C05482=1223.178,35.785,-43.751,-179.162,5.442,148.698
C05483=1223.173,36.035,-43.767,-179.159,5.442,148.697
C05484=1223.168,36.285,-43.783,-179.156,5.443,148.696
C05485=1223.163,36.534,-43.798,-179.154,5.443,148.696
C05486=1223.158,36.784,-43.815,-179.151,5.444,148.695
C05487=1223.154,37.033,-43.830,-179.148,5.444,148.694
C05488=1223.148,37.282,-43.846,-179.146,5.445,148.694
C05489=1223.144,37.532,-43.862,-179.144,5.445,148.693
C05490=1223.138,37.781,-43.878,-179.142,5.446,148.692
C05491=1223.134,38.031,-43.894,-179.139,5.446,148.692
C05492=1223.128,38.280,-43.910,-179.136,5.447,148.691
C05493=1223.123,38.529,-43.926,-179.134,5.447,148.690
C05494=1223.119,38.779,-43.942,-179.131,5.448,148.690
C05495=1223.113,39.028,-43.958,-179.128,5.448,148.689
C05496=1223.108,39.278,-43.974,-179.126,5.449,148.688
C05497=1223.103,39.527,-43.990,-179.124,5.450,148.688
C05498=1223.099,39.777,-44.006,-179.121,5.450,148.687
C05499=1223.093,40.026,-44.022,-179.118,5.451,148.687
C05500=1223.089,40.275,-44.037,-179.116,5.451,148.686
C05501=1223.084,40.525,-44.053,-179.114,5.451,148.685
C05502=1223.079,40.774,-44.070,-179.111,5.452,148.685
C05503=1223.074,41.024,-44.086,-179.108,5.452,148.684
C05504=1223.069,41.273,-44.102,-179.106,5.453,148.683
C05505=1223.064,41.523,-44.118,-179.104,5.454,148.683
C05506=1223.059,41.772,-44.134,-179.101,5.454,148.682
C05507=1223.054,42.022,-44.150,-179.098,5.455,148.681
C05508=1223.049,42.271,-44.166,-179.096,5.455,148.681
C05509=1223.045,42.521,-44.182,-179.093,5.456,148.680
C05510=1223.039,42.770,-44.199,-179.090,5.457,148.679
C05511=1223.035,43.020,-44.215,-179.088,5.457,148.679
C05512=1223.030,43.268,-44.231,-179.085,5.458,148.678
C05513=1223.025,43.519,-44.247,-179.083,5.459,148.678
C05514=1223.019,43.768,-44.264,-179.081,5.458,148.677
C05515=1223.014,44.018,-44.280,-179.078,5.459,148.676
C05516=1223.009,44.267,-44.296,-179.076,5.459,148.676
C05517=1223.005,44.516,-44.313,-179.073,5.460,148.675
C05518=1222.999,44.765,-44.328,-179.070,5.461,148.674
C05519=1222.995,45.015,-44.345,-179.068,5.461,148.674
C05520=1222.989,45.264,-44.361,-179.065,5.462,148.673
C05521=1222.985,45.514,-44.377,-179.063,5.463,148.672
C05522=1222.980,45.763,-44.394,-179.060,5.463,148.672
C05523=1222.975,46.013,-44.410,-179.058,5.464,148.671
C05524=1222.970,46.261,-44.426,-179.055,5.464,148.670
C05525=1222.965,46.512,-44.442,-179.052,5.465,148.670
C05526=1222.960,46.760,-44.458,-179.050,5.465,148.669
C05527=1222.955,47.010,-44.475,-179.047,5.466,148.668
C05528=1222.949,47.260,-44.491,-179.045,5.467,148.668
C05529=1222.945,47.509,-44.508,-179.042,5.467,148.667
C05530=1222.941,47.758,-44.524,-179.040,5.468,148.667
C05531=1222.935,48.008,-44.540,-179.038,5.468,148.666
C05532=1222.931,48.257,-44.557,-179.035,5.468,148.665
C05533=1222.926,48.506,-44.573,-179.032,5.469,148.665
C05534=1222.920,48.756,-44.590,-179.030,5.469,148.664
C05535=1222.915,49.005,-44.606,-179.027,5.470,148.663
C05536=1222.911,49.255,-44.622,-179.025,5.471,148.663
C05537=1222.906,49.504,-44.639,-179.022,5.471,148.662
C05538=1222.901,49.753,-44.655,-179.020,5.472,148.661
C05539=1222.896,50.003,-44.671,-179.017,5.473,148.661
C05540=1222.890,50.252,-44.688,-179.014,5.473,148.660
C05541=1222.886,50.502,-44.705,-179.012,5.474,148.659
C05542=1222.881,50.751,-44.722,-179.010,5.475,148.659
C05543=1222.876,51.001,-44.737,-179.007,5.475,148.658
C05544=1222.872,51.250,-44.754,-179.004,5.476,148.658
C05545=1222.866,51.499,-44.771,-179.002,5.476,148.657
C05546=1222.861,51.749,-44.787,-178.999,5.477,148.656
C05547=1222.857,51.998,-44.804,-178.996,5.477,148.656
C05548=1222.851,52.248,-44.820,-178.994,5.478,148.655
C05549=1222.847,52.497,-44.836,-178.992,5.479,148.655
C05550=1222.842,52.747,-44.854,-178.989,5.479,148.654
C05551=1222.837,52.996,-44.870,-178.986,5.480,148.653
C05552=1222.832,53.245,-44.887,-178.984,5.481,148.653
C05553=1222.828,53.495,-44.903,-178.981,5.481,148.652
C05554=1222.822,53.744,-44.920,-178.978,5.482,148.651
C05555=1222.817,53.994,-44.936,-178.976,5.483,148.651
C05556=1222.812,54.243,-44.952,-178.974,5.483,148.650
C05557=1222.807,54.492,-44.970,-178.971,5.484,148.649
C05558=1222.802,54.742,-44.986,-178.968,5.484,148.649
C05559=1222.797,54.991,-45.003,-178.966,5.485,148.648
C05560=1222.792,55.260,-45.021,-178.963,5.485,148.647
C05561=1222.787,55.527,-45.039,-178.960,5.486,148.647
C05562=1222.782,55.797,-45.056,-178.958,5.487,148.646
C05563=1222.776,56.065,-45.075,-178.955,5.487,148.645
C05564=1222.771,56.314,-45.091,-178.953,5.488,148.645
C05565=1222.767,56.564,-45.108,-178.950,5.488,148.644
C05566=1222.761,56.813,-45.125,-178.948,5.489,148.644
C05567=1222.756,57.062,-45.142,-178.945,5.490,148.643
C05568=1222.752,57.312,-45.158,-178.942,5.490,148.642
C05569=1222.747,57.562,-45.176,-178.940,5.491,148.642
C05570=1222.742,57.810,-45.192,-178.937,5.491,148.641
C05571=1222.736,58.060,-45.209,-178.935,5.492,148.640
C05572=1222.732,58.310,-45.226,-178.932,5.493,148.640
C05573=1222.727,58.558,-45.242,-178.930,5.494,148.639
C05574=1222.722,58.808,-45.259,-178.927,5.494,148.639
C05575=1222.717,59.058,-45.276,-178.925,5.495,148.638
C05576=1222.712,59.308,-45.293,-178.922,5.495,148.637
C05577=1222.707,59.556,-45.310,-178.920,5.496,148.637
C05578=1222.703,59.805,-45.327,-178.917,5.497,148.636
C05579=1222.697,60.055,-45.344,-178.914,5.497,148.635
C05580=1222.693,60.304,-45.361,-178.912,5.498,148.635
C05581=1222.687,60.554,-45.378,-178.909,5.498,148.634
C05582=1222.683,60.803,-45.394,-178.907,5.499,148.633
C05583=1222.677,61.053,-45.412,-178.904,5.500,148.633
C05584=1222.673,61.302,-45.428,-178.902,5.501,148.632
C05585=1222.668,61.551,-45.445,-178.899,5.501,148.632
C05586=1222.663,61.800,-45.463,-178.897,5.502,148.631
C05587=1222.658,62.050,-45.479,-178.894,5.502,148.630
C05588=1222.653,62.300,-45.497,-178.892,5.503,148.630
C05589=1222.649,62.549,-45.513,-178.889,5.504,148.629
C05590=1222.643,62.798,-45.530,-178.886,5.504,148.629
C05591=1222.639,63.047,-45.548,-178.884,5.505,148.628
C05592=1222.633,63.297,-45.565,-178.881,5.505,148.627
C05593=1222.629,63.546,-45.582,-178.879,5.506,148.627
C05594=1222.624,63.796,-45.599,-178.876,5.507,148.626
C05595=1222.619,64.045,-45.615,-178.874,5.508,148.626
C05596=1222.614,64.294,-45.633,-178.871,5.508,148.625
C05597=1222.609,64.544,-45.650,-178.869,5.509,148.624
C05598=1222.604,64.793,-45.667,-178.866,5.510,148.624
C05599=1222.599,65.043,-45.684,-178.863,5.511,148.623
C05600=1222.594,65.291,-45.701,-178.861,5.512,148.622
C05601=1222.589,65.541,-45.719,-178.858,5.512,148.622
C05602=1222.584,65.791,-45.735,-178.855,5.513,148.621
C05603=1222.580,66.040,-45.753,-178.853,5.514,148.621
C05604=1222.575,66.289,-45.770,-178.851,5.514,148.620
C05605=1222.570,66.539,-45.787,-178.848,5.515,148.619
C05606=1222.566,66.788,-45.805,-178.845,5.515,148.619
C05607=1222.560,67.037,-45.821,-178.843,5.516,148.618
C05608=1222.555,67.287,-45.839,-178.841,5.517,148.618
C05609=1222.550,67.536,-45.856,-178.838,5.517,148.617
C05610=1222.545,67.785,-45.873,-178.835,5.518,148.616
C05611=1222.541,68.035,-45.890,-178.833,5.519,148.616
C05612=1222.536,68.284,-45.908,-178.830,5.519,148.615
C05613=1222.531,68.534,-45.925,-178.828,5.520,148.615
C05614=1222.526,68.783,-45.942,-178.825,5.521,148.614
C05615=1222.521,69.032,-45.960,-178.823,5.521,148.613
C05616=1222.515,69.282,-45.977,-178.820,5.522,148.613
C05617=1222.511,69.530,-45.994,-178.818,5.523,148.612
C05618=1222.506,69.780,-46.011,-178.815,5.523,148.611
C05619=1222.501,70.029,-46.029,-178.813,5.524,148.611
C05620=1222.497,70.279,-46.046,-178.809,5.525,148.610
C05621=1222.491,70.529,-46.063,-178.807,5.526,148.609
C05622=1222.486,70.778,-46.081,-178.805,5.527,148.609
C05623=1222.482,71.027,-46.098,-178.802,5.527,148.608
C05624=1222.477,71.277,-46.116,-178.799,5.528,148.608
C05625=1222.471,71.526,-46.133,-178.797,5.529,148.607
C05626=1222.467,71.775,-46.150,-178.795,5.530,148.607
C05627=1222.462,72.024,-46.168,-178.792,5.530,148.606
C05628=1222.457,72.273,-46.186,-178.789,5.531,148.605
C05629=1222.452,72.523,-46.202,-178.787,5.531,148.605
C05630=1222.448,72.772,-46.220,-178.785,5.532,148.604
C05631=1222.442,73.022,-46.237,-178.782,5.533,148.604
C05632=1222.437,73.271,-46.255,-178.779,5.533,148.603
C05633=1222.433,73.520,-46.273,-178.777,5.534,148.602
C05634=1222.428,73.770,-46.290,-178.774,5.535,148.602
C05635=1222.423,74.019,-46.308,-178.771,5.536,148.601
C05636=1222.418,74.269,-46.325,-178.769,5.537,148.601
C05637=1222.414,74.518,-46.343,-178.766,5.537,148.600
C05638=1222.409,74.767,-46.361,-178.763,5.538,148.599
C05639=1222.404,75.017,-46.378,-178.761,5.539,148.599
C05640=1222.399,75.266,-46.396,-178.759,5.540,148.598
C05641=1222.393,75.516,-46.413,-178.756,5.540,148.597
C05642=1222.389,75.764,-46.431,-178.753,5.541,148.597
C05643=1222.384,76.014,-46.449,-178.751,5.542,148.596
C05644=1222.379,76.263,-46.466,-178.749,5.542,148.596
C05645=1222.374,76.513,-46.484,-178.746,5.543,148.595
C05646=1222.369,76.762,-46.502,-178.743,5.543,148.594
C05647=1222.365,77.011,-46.518,-178.741,5.545,148.594
C05648=1222.360,77.260,-46.536,-178.738,5.546,148.593
C05649=1222.355,77.510,-46.554,-178.735,5.546,148.593
C05650=1222.350,77.759,-46.572,-178.733,5.547,148.592
C05651=1222.345,78.009,-46.590,-178.731,5.548,148.592
C05652=1222.340,78.258,-46.608,-178.728,5.548,148.591
C05653=1222.335,78.507,-46.626,-178.725,5.549,148.590
C05654=1222.331,78.756,-46.642,-178.723,5.550,148.590
C05655=1222.326,79.006,-46.660,-178.721,5.551,148.589
C05656=1222.321,79.255,-46.678,-178.718,5.551,148.589
C05657=1222.316,79.504,-46.696,-178.715,5.553,148.588
C05658=1222.311,79.754,-46.713,-178.712,5.553,148.587
C05659=1222.306,80.003,-46.731,-178.710,5.554,148.587
C05660=1222.301,80.252,-46.749,-178.708,5.555,148.586
C05661=1222.296,80.501,-46.767,-178.705,5.555,148.585
C05662=1222.291,80.750,-46.785,-178.703,5.556,148.585
C05663=1222.286,81.001,-46.803,-178.700,5.557,148.584
C05664=1222.281,81.268,-46.822,-178.697,5.558,148.584
C05665=1222.276,81.537,-46.841,-178.694,5.559,148.583
C05666=1222.271,81.805,-46.861,-178.692,5.559,148.582
C05667=1222.265,82.074,-46.880,-178.689,5.560,148.582
C05668=1222.260,82.323,-46.898,-178.686,5.561,148.581
C05669=1222.255,82.572,-46.916,-178.684,5.562,148.581
C05670=1222.251,82.822,-46.934,-178.681,5.563,148.580
C05671=1222.246,83.071,-46.952,-178.678,5.564,148.579
C05672=1222.241,83.320,-46.970,-178.676,5.564,148.579
C05673=1222.236,83.570,-46.988,-178.674,5.565,148.578
C05674=1222.231,83.819,-47.006,-178.671,5.566,148.578
C05675=1222.226,84.068,-47.024,-178.668,5.566,148.577
C05676=1222.222,84.317,-47.042,-178.666,5.567,148.577
C05677=1222.216,84.567,-47.059,-178.663,5.569,148.576
C05678=1222.212,84.817,-47.077,-178.661,5.569,148.575
C05679=1222.207,85.066,-47.095,-178.658,5.570,148.575
C05680=1222.202,85.315,-47.113,-178.656,5.571,148.574
C05681=1222.197,85.564,-47.131,-178.653,5.571,148.574
C05682=1222.192,85.814,-47.149,-178.651,5.572,148.573
C05683=1222.187,86.063,-47.167,-178.648,5.573,148.572
C05684=1222.183,86.312,-47.185,-178.645,5.574,148.572
C05685=1222.178,86.562,-47.204,-178.643,5.575,148.571
C05686=1222.173,86.811,-47.222,-178.640,5.575,148.571
C05687=1222.168,87.060,-47.240,-178.638,5.576,148.570
C05688=1222.163,87.309,-47.258,-178.635,5.577,148.569
C05689=1222.159,87.558,-47.276,-178.633,5.578,148.569
C05690=1222.154,87.807,-47.294,-178.630,5.579,148.568
C05691=1222.150,88.057,-47.313,-178.627,5.580,148.568
C05692=1222.144,88.306,-47.331,-178.625,5.581,148.567
C05693=1222.139,88.556,-47.349,-178.623,5.581,148.567
C05694=1222.134,88.805,-47.367,-178.620,5.582,148.566
C05695=1222.129,89.054,-47.385,-178.617,5.583,148.565
C05696=1222.125,89.304,-47.403,-178.615,5.583,148.565
C05697=1222.120,89.553,-47.421,-178.612,5.585,148.564
C05698=1222.115,89.802,-47.439,-178.609,5.586,148.564
C05699=1222.110,90.051,-47.459,-178.607,5.586,148.563
C05700=1222.105,90.300,-47.477,-178.605,5.587,148.563
C05701=1222.101,90.550,-47.495,-178.602,5.588,148.562
C05702=1222.096,90.799,-47.513,-178.599,5.588,148.561
C05703=1222.091,91.048,-47.531,-178.597,5.590,148.561
C05704=1222.086,91.298,-47.549,-178.594,5.591,148.560
C05705=1222.081,91.547,-47.569,-178.591,5.591,148.560
C05706=1222.076,91.796,-47.587,-178.589,5.592,148.559
C05707=1222.071,92.045,-47.605,-178.587,5.593,148.558
C05708=1222.066,92.295,-47.623,-178.584,5.593,148.558
C05709=1222.062,92.545,-47.641,-178.581,5.595,148.557
C05710=1222.057,92.793,-47.660,-178.579,5.596,148.557
C05711=1222.052,93.043,-47.678,-178.576,5.596,148.556
C05712=1222.047,93.292,-47.696,-178.574,5.597,148.556
C05713=1222.043,93.542,-47.714,-178.571,5.598,148.555
C05714=1222.037,93.790,-47.734,-178.569,5.599,148.554
C05715=1222.032,94.040,-47.752,-178.566,5.600,148.554
C05716=1222.028,94.290,-47.770,-178.563,5.601,148.553
C05717=1222.023,94.538,-47.789,-178.561,5.602,148.553
C05718=1222.018,94.788,-47.807,-178.558,5.602,148.552
C05719=1222.013,95.037,-47.825,-178.556,5.603,148.552
C05720=1222.009,95.286,-47.844,-178.553,5.604,148.551
C05721=1222.004,95.535,-47.862,-178.550,5.605,148.550
C05722=1221.998,95.785,-47.881,-178.548,5.606,148.550
C05723=1221.994,96.034,-47.900,-178.545,5.607,148.549
C05724=1221.989,96.283,-47.918,-178.543,5.607,148.549
C05725=1221.984,96.533,-47.937,-178.540,5.609,148.548
C05726=1221.980,96.782,-47.956,-178.538,5.610,148.548
C05727=1221.975,97.031,-47.974,-178.535,5.611,148.547
C05728=1221.969,97.280,-47.993,-178.533,5.611,148.546
C05729=1221.965,97.530,-48.011,-178.530,5.612,148.546
C05730=1221.960,97.779,-48.029,-178.527,5.614,148.545
C05731=1221.955,98.028,-48.049,-178.525,5.614,148.545
C05732=1221.951,98.278,-48.067,-178.522,5.615,148.544
C05733=1221.946,98.526,-48.086,-178.520,5.616,148.544
C05734=1221.940,98.776,-48.104,-178.517,5.616,148.543
C05735=1221.936,99.025,-48.123,-178.514,5.618,148.542
C05736=1221.931,99.274,-48.141,-178.512,5.619,148.542
C05737=1221.926,99.523,-48.160,-178.510,5.619,148.541
C05738=1221.922,99.773,-48.179,-178.507,5.620,148.541
C05739=1221.916,100.022,-48.198,-178.505,5.621,148.540
C05740=1221.912,100.272,-48.216,-178.502,5.622,148.540
C05741=1221.907,100.520,-48.235,-178.499,5.623,148.539
C05742=1221.902,100.770,-48.254,-178.497,5.624,148.539
C05743=1221.898,101.019,-48.273,-178.494,5.624,148.538
C05744=1221.892,101.268,-48.291,-178.492,5.626,148.538
C05745=1221.888,101.518,-48.310,-178.489,5.627,148.537
C05746=1221.883,101.767,-48.329,-178.486,5.627,148.536
C05747=1221.878,102.016,-48.348,-178.484,5.628,148.536
C05748=1221.874,102.265,-48.367,-178.482,5.629,148.535
C05749=1221.868,102.514,-48.385,-178.478,5.630,148.535
C05750=1221.864,102.764,-48.404,-178.476,5.631,148.534
C05751=1221.859,103.013,-48.423,-178.474,5.632,148.533
C05752=1221.854,103.262,-48.442,-178.471,5.633,148.533
C05753=1221.849,103.511,-48.461,-178.468,5.634,148.532
C05754=1221.844,103.761,-48.479,-178.466,5.635,148.532
C05755=1221.840,104.010,-48.499,-178.464,5.636,148.531
C05756=1221.835,104.259,-48.518,-178.461,5.637,148.531
C05757=1221.830,104.509,-48.537,-178.458,5.638,148.530
C05758=1221.825,104.757,-48.555,-178.456,5.639,148.530
C05759=1221.821,105.007,-48.575,-178.453,5.639,148.529
C05760=1221.816,105.256,-48.593,-178.450,5.640,148.528
C05761=1221.810,105.505,-48.612,-178.448,5.642,148.528
C05762=1221.806,105.755,-48.632,-178.445,5.642,148.527
C05763=1221.801,106.004,-48.650,-178.443,5.643,148.527
C05764=1221.796,106.253,-48.669,-178.440,5.644,148.526
C05765=1221.791,106.502,-48.688,-178.437,5.645,148.526
C05766=1221.787,106.751,-48.708,-178.435,5.646,148.525
C05767=1221.782,107.001,-48.726,-178.433,5.647,148.525
C05768=1221.777,107.269,-48.747,-178.430,5.648,148.524
C05769=1221.771,107.537,-48.768,-178.427,5.649,148.524
C05770=1221.766,107.806,-48.788,-178.425,5.650,148.523
C05771=1221.761,108.074,-48.809,-178.421,5.651,148.522
C05772=1221.757,108.324,-48.828,-178.419,5.652,148.522
C05773=1221.751,108.573,-48.847,-178.417,5.653,148.521
C05774=1221.747,108.822,-48.865,-178.414,5.654,148.521
C05775=1221.742,109.071,-48.885,-178.411,5.655,148.520
C05776=1221.737,109.321,-48.904,-178.409,5.656,148.520
C05777=1221.732,109.569,-48.923,-178.406,5.657,148.519
C05778=1221.727,109.819,-48.943,-178.403,5.658,148.518
C05779=1221.723,110.069,-48.962,-178.401,5.659,148.518
C05780=1221.718,110.317,-48.981,-178.399,5.660,148.517
C05781=1221.713,110.567,-49.001,-178.396,5.661,148.517
C05782=1221.708,110.816,-49.019,-178.393,5.662,148.516
C05783=1221.704,111.065,-49.038,-178.391,5.663,148.516
C05784=1221.698,111.314,-49.058,-178.388,5.664,148.515
C05785=1221.694,111.564,-49.077,-178.386,5.665,148.515
C05786=1221.689,111.812,-49.096,-178.383,5.666,148.514
C05787=1221.684,112.062,-49.116,-178.380,5.667,148.513
C05788=1221.679,112.312,-49.135,-178.378,5.668,148.513
C05789=1221.675,112.560,-49.154,-178.375,5.669,148.512
C05790=1221.670,112.810,-49.174,-178.373,5.670,148.512
C05791=1221.665,113.059,-49.193,-178.370,5.671,148.511
C05792=1221.660,113.308,-49.213,-178.368,5.672,148.511
C05793=1221.655,113.557,-49.231,-178.365,5.673,148.510
C05794=1221.651,113.806,-49.251,-178.362,5.674,148.510
C05795=1221.646,114.056,-49.271,-178.360,5.675,148.509
C05796=1221.641,114.305,-49.290,-178.357,5.676,148.509
C05797=1221.637,114.554,-49.309,-178.355,5.677,148.508
C05798=1221.632,114.804,-49.329,-178.352,5.678,148.508
C05799=1221.627,115.052,-49.348,-178.350,5.679,148.507
C05800=1221.622,115.302,-49.368,-178.347,5.680,148.506
C05801=1221.616,115.551,-49.387,-178.344,5.681,148.506
C05802=1221.612,115.800,-49.406,-178.342,5.682,148.505
C05803=1221.608,116.050,-49.426,-178.339,5.683,148.505
C05804=1221.602,116.299,-49.445,-178.337,5.684,148.504
C05805=1221.598,116.547,-49.465,-178.334,5.685,148.504
C05806=1221.593,116.797,-49.485,-178.332,5.686,148.503
C05807=1221.588,117.046,-49.504,-178.329,5.687,148.503
C05808=1221.584,117.295,-49.523,-178.326,5.688,148.502
C05809=1221.579,117.545,-49.543,-178.324,5.689,148.502
C05810=1221.574,117.794,-49.562,-178.321,5.690,148.501
C05811=1221.569,118.043,-49.582,-178.319,5.691,148.501
C05812=1221.565,118.292,-49.602,-178.316,5.692,148.500
C05813=1221.559,118.541,-49.622,-178.314,5.693,148.500
C05814=1221.554,118.791,-49.641,-178.311,5.694,148.499
C05815=1221.550,119.040,-49.660,-178.308,5.696,148.499
C05816=1221.545,119.289,-49.680,-178.306,5.696,148.498
C05817=1221.541,119.538,-49.700,-178.304,5.697,148.498
C05818=1221.536,119.787,-49.720,-178.301,5.699,148.497
C05819=1221.531,120.036,-49.739,-178.298,5.699,148.496
C05820=1221.526,120.286,-49.758,-178.296,5.700,148.496
C05821=1221.521,120.535,-49.779,-178.293,5.702,148.495
C05822=1221.516,120.783,-49.798,-178.291,5.703,148.495
C05823=1221.511,121.033,-49.818,-178.288,5.703,148.494
C05824=1221.507,121.283,-49.837,-178.285,5.705,148.494
C05825=1221.502,121.532,-49.858,-178.283,5.706,148.493
C05826=1221.497,121.780,-49.877,-178.281,5.707,148.493
C05827=1221.492,122.030,-49.897,-178.277,5.708,148.492
C05828=1221.488,122.279,-49.917,-178.275,5.709,148.492
C05829=1221.484,122.528,-49.936,-178.273,5.710,148.491
C05830=1221.478,122.777,-49.956,-178.270,5.712,148.491
C05831=1221.474,123.026,-49.976,-178.267,5.712,148.490
C05832=1221.469,123.276,-49.996,-178.265,5.713,148.490
C05833=1221.465,123.524,-50.016,-178.262,5.715,148.489
C05834=1221.459,123.773,-50.035,-178.260,5.716,148.489
C05835=1221.455,124.023,-50.055,-178.257,5.716,148.488
C05836=1221.450,124.272,-50.075,-178.254,5.718,148.487
C05837=1221.445,124.521,-50.095,-178.252,5.719,148.487
C05838=1221.440,124.770,-50.115,-178.249,5.719,148.486
C05839=1221.435,125.020,-50.135,-178.247,5.721,148.486
C05840=1221.430,125.269,-50.155,-178.244,5.722,148.485
C05841=1221.426,125.518,-50.175,-178.241,5.724,148.485
C05842=1221.421,125.768,-50.195,-178.239,5.724,148.484
C05843=1221.416,126.016,-50.215,-178.237,5.725,148.484
C05844=1221.411,126.265,-50.234,-178.234,5.727,148.483
C05845=1221.407,126.514,-50.255,-178.231,5.728,148.483
C05846=1221.402,126.764,-50.275,-178.229,5.728,148.482
C05847=1221.398,127.013,-50.295,-178.226,5.730,148.482
C05848=1221.392,127.262,-50.314,-178.224,5.731,148.481
C05849=1221.388,127.511,-50.335,-178.221,5.732,148.481
C05850=1221.383,127.760,-50.354,-178.218,5.733,148.480
C05851=1221.379,128.009,-50.375,-178.216,5.734,148.480
C05852=1221.373,128.259,-50.395,-178.213,5.735,148.479
C05853=1221.369,128.508,-50.415,-178.211,5.736,148.479
C05854=1221.364,128.756,-50.435,-178.208,5.737,148.478
C05855=1221.359,129.006,-50.455,-178.206,5.739,148.478
C05856=1221.354,129.255,-50.475,-178.203,5.739,148.477
C05857=1221.350,129.504,-50.495,-178.200,5.741,148.477
C05858=1221.345,129.753,-50.515,-178.198,5.742,148.476
C05859=1221.340,130.003,-50.536,-178.196,5.743,148.476
C05860=1221.335,130.252,-50.556,-178.192,5.744,148.475
C05861=1221.331,130.501,-50.576,-178.190,5.745,148.475
C05862=1221.326,130.750,-50.596,-178.188,5.746,148.474
C05863=1221.321,130.999,-50.616,-178.185,5.748,148.474
C05864=1221.317,131.248,-50.636,-178.182,5.748,148.473
C05865=1221.311,131.498,-50.657,-178.180,5.750,148.473
C05866=1221.307,131.747,-50.677,-178.178,5.751,148.472
C05867=1221.302,131.996,-50.697,-178.175,5.752,148.472
C05868=1221.298,132.245,-50.718,-178.172,5.754,148.471
C05869=1221.292,132.495,-50.738,-178.170,5.754,148.471
C05870=1221.288,132.743,-50.758,-178.167,5.756,148.470
C05871=1221.283,132.992,-50.778,-178.165,5.757,148.470
C05872=1221.278,133.261,-50.800,-178.162,5.758,148.469
C05873=1221.273,133.529,-50.822,-178.159,5.759,148.469
C05874=1221.268,133.798,-50.844,-178.156,5.760,148.468
C05875=1221.262,134.067,-50.866,-178.154,5.761,148.467
C05876=1221.258,134.316,-50.887,-178.151,5.763,148.467
C05877=1221.253,134.565,-50.906,-178.149,5.764,148.466
C05878=1221.248,134.815,-50.927,-178.146,5.765,148.466
C05879=1221.244,135.063,-50.948,-178.143,5.766,148.465
C05880=1221.239,135.312,-50.968,-178.140,5.768,148.465
C05881=1221.234,135.562,-50.989,-178.138,5.769,148.464
C05882=1221.229,135.811,-51.009,-178.136,5.769,148.464
C05883=1221.225,136.060,-51.029,-178.133,5.771,148.463
C05884=1221.220,136.309,-51.049,-178.130,5.772,148.463
C05885=1221.215,136.558,-51.070,-178.128,5.774,148.462
C05886=1221.211,136.807,-51.091,-178.125,5.775,148.462
C05887=1221.205,137.057,-51.112,-178.122,5.776,148.461
C05888=1221.201,137.306,-51.132,-178.120,5.777,148.461
C05889=1221.197,137.554,-51.152,-178.118,5.778,148.460
C05890=1221.191,137.804,-51.173,-178.115,5.779,148.460
C05891=1221.187,138.053,-51.194,-178.112,5.780,148.459
C05892=1221.182,138.302,-51.213,-178.110,5.782,148.459
C05893=1221.177,138.552,-51.234,-178.107,5.783,148.458
C05894=1221.173,138.800,-51.255,-178.104,5.784,148.458
C05895=1221.167,139.050,-51.276,-178.102,5.785,148.458
C05896=1221.163,139.299,-51.296,-178.100,5.786,148.457
C05897=1221.159,139.548,-51.316,-178.097,5.788,148.457
C05898=1221.153,139.797,-51.337,-178.094,5.788,148.456
C05899=1221.149,140.046,-51.358,-178.092,5.790,148.456
C05900=1221.144,140.295,-51.379,-178.089,5.791,148.455
C05901=1221.139,140.544,-51.399,-178.086,5.793,148.455
C05902=1221.134,140.793,-51.420,-178.084,5.794,148.454
C05903=1221.130,141.042,-51.440,-178.081,5.795,148.454
C05904=1221.125,141.291,-51.461,-178.079,5.796,148.453
C05905=1221.120,141.540,-51.482,-178.076,5.797,148.453
C05906=1221.116,141.789,-51.503,-178.074,5.798,148.452
C05907=1221.111,142.038,-51.524,-178.071,5.799,148.452
C05908=1221.106,142.287,-51.544,-178.069,5.801,148.451
C05909=1221.101,142.536,-51.565,-178.066,5.802,148.451
C05910=1221.097,142.785,-51.586,-178.063,5.803,148.450
C05911=1221.092,143.035,-51.607,-178.061,5.804,148.450
C05912=1221.088,143.284,-51.627,-178.058,5.806,148.449
C05913=1221.083,143.533,-51.648,-178.056,5.807,148.449
C05914=1221.078,143.782,-51.669,-178.053,5.809,148.448
C05915=1221.073,144.031,-51.690,-178.051,5.809,148.448
C05916=1221.068,144.280,-51.711,-178.048,5.811,148.447
C05917=1221.064,144.529,-51.732,-178.045,5.812,148.447
C05918=1221.059,144.778,-51.753,-178.043,5.813,148.446
C05919=1221.054,145.027,-51.773,-178.040,5.814,148.446
C05920=1221.049,145.276,-51.795,-178.037,5.816,148.445
C05921=1221.045,145.526,-51.815,-178.035,5.817,148.445
C05922=1221.040,145.775,-51.836,-178.032,5.818,148.444
C05923=1221.036,146.024,-51.857,-178.030,5.819,148.444
C05924=1221.031,146.273,-51.878,-178.028,5.820,148.444
C05925=1221.026,146.522,-51.899,-178.025,5.822,148.443
C05926=1221.021,146.771,-51.920,-178.023,5.823,148.443
C05927=1221.016,147.020,-51.941,-178.019,5.824,148.442
C05928=1221.012,147.269,-51.963,-178.017,5.825,148.442
C05929=1221.007,147.518,-51.983,-178.015,5.827,148.441
C05930=1221.002,147.768,-52.004,-178.012,5.828,148.441
C05931=1220.998,148.016,-52.025,-178.009,5.829,148.440
C05932=1220.993,148.265,-52.046,-178.007,5.830,148.440
C05933=1220.988,148.514,-52.067,-178.004,5.832,148.439
C05934=1220.984,148.763,-52.089,-178.002,5.833,148.439
C05935=1220.979,149.013,-52.110,-177.999,5.834,148.438
C05936=1220.974,149.262,-52.130,-177.997,5.835,148.438
C05937=1220.970,149.510,-52.152,-177.994,5.837,148.437
C05938=1220.965,149.760,-52.173,-177.992,5.838,148.437
C05939=1220.960,150.009,-52.194,-177.989,5.840,148.436
C05940=1220.955,150.258,-52.216,-177.986,5.840,148.436
C05941=1220.951,150.507,-52.236,-177.984,5.842,148.435
C05942=1220.946,150.756,-52.258,-177.982,5.843,148.435
C05943=1220.941,151.005,-52.279,-177.978,5.845,148.434
C05944=1220.937,151.254,-52.300,-177.976,5.846,148.434
C05945=1220.932,151.503,-52.321,-177.974,5.847,148.434
C05946=1220.927,151.752,-52.343,-177.970,5.849,148.433
C05947=1220.922,152.001,-52.364,-177.968,5.850,148.433
C05948=1220.918,152.251,-52.384,-177.965,5.851,148.432
C05949=1220.913,152.499,-52.406,-177.963,5.852,148.432
C05950=1220.908,152.749,-52.427,-177.960,5.854,148.431
C05951=1220.903,152.997,-52.449,-177.958,5.855,148.431
C05952=1220.900,153.246,-52.470,-177.955,5.856,148.430
C05953=1220.894,153.496,-52.491,-177.953,5.857,148.430
C05954=1220.890,153.744,-52.513,-177.950,5.859,148.429
C05955=1220.884,153.994,-52.534,-177.948,5.860,148.429
C05956=1220.880,154.243,-52.556,-177.945,5.862,148.429
C05957=1220.875,154.492,-52.577,-177.943,5.862,148.428
C05958=1220.871,154.740,-52.598,-177.940,5.864,148.428
C05959=1220.866,154.990,-52.619,-177.938,5.865,148.427
C05960=1220.861,155.239,-52.641,-177.935,5.867,148.427
C05961=1220.857,155.488,-52.663,-177.932,5.868,148.426
C05962=1220.851,155.737,-52.684,-177.930,5.869,148.426
C05963=1220.847,155.986,-52.706,-177.927,5.871,148.425
C05964=1220.843,156.235,-52.727,-177.925,5.872,148.425
C05965=1220.838,156.484,-52.748,-177.922,5.874,148.424
C05966=1220.833,156.733,-52.770,-177.919,5.874,148.424
C05967=1220.829,156.982,-52.791,-177.917,5.876,148.423
C05968=1220.823,157.231,-52.812,-177.915,5.877,148.423
C05969=1220.819,157.480,-52.834,-177.911,5.879,148.422
C05970=1220.814,157.729,-52.856,-177.909,5.880,148.422
C05971=1220.809,157.978,-52.877,-177.907,5.881,148.422
C05972=1220.804,158.227,-52.899,-177.903,5.883,148.421
C05973=1220.800,158.476,-52.921,-177.901,5.884,148.421
C05974=1220.796,158.725,-52.941,-177.899,5.886,148.420
C05975=1220.791,158.975,-52.963,-177.896,5.886,148.420
C05976=1220.786,159.243,-52.987,-177.893,5.888,148.419
C05977=1220.781,159.513,-53.011,-177.890,5.890,148.419
C05978=1220.776,159.782,-53.033,-177.888,5.892,148.418
C05979=1220.771,160.051,-53.057,-177.885,5.892,148.418
C05980=1220.766,160.300,-53.078,-177.882,5.894,148.417
C05981=1220.761,160.548,-53.100,-177.880,5.896,148.417
C05982=1220.756,160.798,-53.122,-177.877,5.896,148.416
C05983=1220.752,161.046,-53.144,-177.874,5.898,148.416
C05984=1220.747,161.296,-53.166,-177.872,5.899,148.416
C05985=1220.742,161.544,-53.188,-177.869,5.901,148.415
C05986=1220.737,161.794,-53.209,-177.867,5.902,148.415
C05987=1220.733,162.043,-53.231,-177.864,5.904,148.414
C05988=1220.728,162.292,-53.252,-177.862,5.905,148.414
C05989=1220.724,162.541,-53.274,-177.859,5.906,148.413
C05990=1220.719,162.790,-53.296,-177.857,5.908,148.413
C05991=1220.714,163.038,-53.318,-177.854,5.909,148.413
C05992=1220.710,163.288,-53.340,-177.851,5.910,148.412
C05993=1220.705,163.536,-53.361,-177.849,5.912,148.412
C05994=1220.701,163.786,-53.383,-177.847,5.913,148.411
C05995=1220.696,164.034,-53.405,-177.844,5.915,148.411
C05996=1220.692,164.284,-53.427,-177.841,5.916,148.410
C05997=1220.687,164.532,-53.449,-177.839,5.917,148.410
C05998=1220.682,164.782,-53.471,-177.836,5.919,148.409
C05999=1220.677,165.031,-53.493,-177.833,5.920,148.409
C06000=1220.672,165.279,-53.515,-177.831,5.922,148.408
C06001=1220.668,165.528,-53.537,-177.829,5.923,148.408
C06002=1220.663,165.777,-53.559,-177.826,5.925,148.408
C06003=1220.658,166.026,-53.581,-177.823,5.926,148.407
C06004=1220.654,166.275,-53.602,-177.821,5.927,148.407
C06005=1220.649,166.524,-53.624,-177.818,5.929,148.406
C06006=1220.644,166.773,-53.646,-177.815,5.929,148.406
C06007=1220.639,167.023,-53.669,-177.813,5.931,148.405
C06008=1220.635,167.271,-53.690,-177.810,5.933,148.405
C06009=1220.630,167.521,-53.712,-177.808,5.934,148.405
C06010=1220.625,167.769,-53.734,-177.805,5.936,148.404
C06011=1220.621,168.019,-53.756,-177.802,5.937,148.404
C06012=1220.616,168.267,-53.778,-177.800,5.938,148.403
C06013=1220.612,168.516,-53.801,-177.797,5.940,148.403
C06014=1220.607,168.765,-53.823,-177.795,5.941,148.402
C06015=1220.603,169.014,-53.845,-177.792,5.943,148.402
C06016=1220.598,169.263,-53.867,-177.790,5.945,148.402
C06017=1220.593,169.512,-53.889,-177.787,5.946,148.401
C06018=1220.588,169.761,-53.911,-177.784,5.947,148.401
C06019=1220.584,170.010,-53.934,-177.782,5.949,148.400
C06020=1220.580,170.259,-53.956,-177.780,5.950,148.400
C06021=1220.575,170.508,-53.977,-177.777,5.952,148.400
C06022=1220.570,170.758,-54.000,-177.774,5.952,148.399
C06023=1220.565,171.006,-54.022,-177.772,5.954,148.399
C06024=1220.561,171.255,-54.045,-177.769,5.956,148.398
C06025=1220.555,171.504,-54.067,-177.767,5.957,148.398
C06026=1220.551,171.753,-54.089,-177.764,5.958,148.397
C06027=1220.546,172.002,-54.111,-177.761,5.960,148.397
C06028=1220.542,172.251,-54.133,-177.759,5.961,148.396
C06029=1220.537,172.500,-54.156,-177.756,5.963,148.396
C06030=1220.532,172.749,-54.178,-177.753,5.965,148.396
C06031=1220.528,172.998,-54.200,-177.751,5.966,148.395
C06032=1220.523,173.247,-54.223,-177.748,5.967,148.395
C06033=1220.518,173.496,-54.245,-177.746,5.969,148.394
C06034=1220.514,173.745,-54.268,-177.743,5.970,148.394
C06035=1220.509,173.994,-54.290,-177.741,5.972,148.393
C06036=1220.505,174.243,-54.312,-177.738,5.974,148.393
C06037=1220.500,174.491,-54.334,-177.736,5.975,148.393
C06038=1220.495,174.741,-54.357,-177.733,5.976,148.392
C06039=1220.491,174.989,-54.380,-177.730,5.978,148.392
C06040=1220.485,175.238,-54.402,-177.728,5.979,148.391
C06041=1220.481,175.488,-54.424,-177.725,5.981,148.391
C06042=1220.477,175.736,-54.447,-177.723,5.982,148.391
C06043=1220.472,175.985,-54.469,-177.720,5.983,148.390
C06044=1220.468,176.234,-54.492,-177.717,5.985,148.390
C06045=1220.463,176.484,-54.514,-177.715,5.987,148.389
C06046=1220.458,176.732,-54.537,-177.713,5.988,148.389
C06047=1220.453,176.981,-54.559,-177.710,5.990,148.389
C06048=1220.449,177.230,-54.582,-177.707,5.991,148.388
C06049=1220.444,177.479,-54.604,-177.705,5.992,148.388
C06050=1220.440,177.728,-54.627,-177.702,5.994,148.387
C06051=1220.435,177.977,-54.649,-177.699,5.996,148.387
C06052=1220.430,178.225,-54.672,-177.697,5.997,148.387
C06053=1220.426,178.475,-54.694,-177.694,5.998,148.386
C06054=1220.421,178.724,-54.718,-177.692,6.000,148.386
C06055=1220.416,178.972,-54.739,-177.689,6.001,148.385
C06056=1220.411,179.222,-54.763,-177.687,6.003,148.385
C06057=1220.407,179.470,-54.786,-177.684,6.005,148.385
C06058=1220.402,179.719,-54.808,-177.681,6.006,148.384
C06059=1220.398,179.968,-54.831,-177.679,6.007,148.384
C06060=1220.393,180.218,-54.853,-177.676,6.009,148.383
C06061=1220.389,180.466,-54.876,-177.674,6.011,148.383
C06062=1220.384,180.715,-54.899,-177.672,6.012,148.382
C06063=1220.379,180.964,-54.921,-177.669,6.014,148.382
C06064=1220.375,181.213,-54.944,-177.666,6.015,148.382
C06065=1220.371,181.462,-54.967,-177.664,6.016,148.381
C06066=1220.365,181.711,-54.989,-177.661,6.018,148.381
C06067=1220.360,181.960,-55.013,-177.658,6.020,148.380
C06068=1220.356,182.208,-55.036,-177.656,6.022,148.380
C06069=1220.351,182.458,-55.058,-177.653,6.022,148.379
C06070=1220.347,182.706,-55.081,-177.650,6.024,148.379
C06071=1220.342,182.955,-55.104,-177.648,6.026,148.379
C06072=1220.338,183.204,-55.127,-177.646,6.027,148.378
C06073=1220.333,183.453,-55.149,-177.643,6.029,148.378
C06074=1220.328,183.702,-55.172,-177.640,6.031,148.378
C06075=1220.324,183.951,-55.195,-177.637,6.032,148.377
C06076=1220.319,184.200,-55.218,-177.635,6.033,148.377
C06077=1220.314,184.449,-55.241,-177.633,6.035,148.376
C06078=1220.310,184.698,-55.264,-177.630,6.037,148.376
C06079=1220.305,184.946,-55.287,-177.627,6.039,148.376
C06080=1220.300,185.216,-55.312,-177.624,6.040,148.375
C06081=1220.295,185.485,-55.336,-177.622,6.041,148.375
C06082=1220.290,185.756,-55.362,-177.619,6.043,148.374
C06083=1220.286,186.025,-55.386,-177.616,6.045,148.374
C06084=1220.280,186.274,-55.409,-177.614,6.046,148.373
C06085=1220.276,186.523,-55.433,-177.611,6.048,148.373
C06086=1220.271,186.772,-55.456,-177.608,6.050,148.373
C06087=1220.267,187.021,-55.479,-177.606,6.051,148.372
C06088=1220.262,187.270,-55.502,-177.604,6.053,148.372
C06089=1220.258,187.519,-55.525,-177.601,6.055,148.372
C06090=1220.253,187.767,-55.548,-177.598,6.056,148.371
C06091=1220.248,188.016,-55.571,-177.596,6.057,148.371
C06092=1220.244,188.265,-55.594,-177.593,6.059,148.370
C06093=1220.239,188.514,-55.617,-177.590,6.061,148.370
C06094=1220.235,188.763,-55.640,-177.588,6.063,148.370
C06095=1220.230,189.012,-55.663,-177.586,6.064,148.369
C06096=1220.225,189.261,-55.687,-177.583,6.066,148.369
C06097=1220.220,189.509,-55.710,-177.580,6.067,148.368
C06098=1220.215,189.758,-55.733,-177.577,6.069,148.368
C06099=1220.211,190.007,-55.756,-177.575,6.070,148.368
C06100=1220.207,190.256,-55.779,-177.572,6.072,148.367
C06101=1220.202,190.505,-55.803,-177.570,6.074,148.367
C06102=1220.198,190.754,-55.827,-177.567,6.075,148.367
C06103=1220.193,191.003,-55.850,-177.565,6.077,148.366
C06104=1220.189,191.251,-55.873,-177.562,6.078,148.366
C06105=1220.184,191.500,-55.896,-177.559,6.080,148.365
C06106=1220.180,191.749,-55.919,-177.557,6.082,148.365
C06107=1220.175,191.999,-55.943,-177.554,6.083,148.365
C06108=1220.170,192.247,-55.966,-177.552,6.084,148.364
C06109=1220.165,192.496,-55.989,-177.549,6.086,148.364
C06110=1220.160,192.745,-56.012,-177.547,6.088,148.364
C06111=1220.156,192.993,-56.036,-177.544,6.090,148.363
C06112=1220.152,193.242,-56.059,-177.541,6.092,148.363
C06113=1220.147,193.491,-56.083,-177.539,6.093,148.362
C06114=1220.142,193.740,-56.106,-177.536,6.094,148.362
C06115=1220.138,193.989,-56.129,-177.534,6.096,148.362
C06116=1220.133,194.238,-56.153,-177.531,6.098,148.361
C06117=1220.129,194.487,-56.177,-177.529,6.099,148.361
C06118=1220.124,194.736,-56.200,-177.526,6.101,148.360
C06119=1220.119,194.985,-56.223,-177.523,6.103,148.360
C06120=1220.114,195.234,-56.247,-177.521,6.105,148.360
C06121=1220.110,195.482,-56.271,-177.518,6.106,148.359
C06122=1220.105,195.731,-56.294,-177.516,6.107,148.359
C06123=1220.101,195.980,-56.318,-177.513,6.109,148.359
C06124=1220.096,196.229,-56.341,-177.511,6.111,148.358
C06125=1220.092,196.478,-56.365,-177.508,6.113,148.358
C06126=1220.087,196.727,-56.388,-177.505,6.114,148.357
C06127=1220.082,196.976,-56.412,-177.502,6.116,148.357
C06128=1220.078,197.224,-56.436,-177.500,6.117,148.357
C06129=1220.073,197.473,-56.459,-177.498,6.119,148.356
C06130=1220.068,197.722,-56.483,-177.495,6.121,148.356
C06131=1220.064,197.971,-56.507,-177.492,6.123,148.356
C06132=1220.059,198.220,-56.530,-177.490,6.125,148.355
C06133=1220.055,198.469,-56.553,-177.488,6.126,148.355
C06134=1220.050,198.717,-56.577,-177.485,6.127,148.355
C06135=1220.046,198.966,-56.601,-177.482,6.129,148.354
C06136=1220.041,199.214,-56.625,-177.480,6.131,148.354
C06137=1220.036,199.464,-56.648,-177.477,6.133,148.354
C06138=1220.032,199.713,-56.672,-177.474,6.135,148.353
C06139=1220.027,199.961,-56.696,-177.472,6.136,148.353
C06140=1220.023,200.210,-56.719,-177.469,6.137,148.352
C06141=1220.019,200.459,-56.743,-177.467,6.139,148.352
C06142=1220.014,200.708,-56.767,-177.464,6.141,148.352
C06143=1220.010,200.957,-56.791,-177.461,6.143,148.351
C06144=1220.004,201.206,-56.815,-177.459,6.145,148.351
C06145=1220.000,201.454,-56.839,-177.457,6.146,148.351
C06146=1219.995,201.703,-56.862,-177.454,6.148,148.350
C06147=1219.991,201.952,-56.886,-177.451,6.149,148.350
C06148=1219.986,202.201,-56.910,-177.449,6.151,148.350
C06149=1219.982,202.449,-56.934,-177.446,6.153,148.349
C06150=1219.977,202.698,-56.958,-177.443,6.155,148.349
C06151=1219.973,202.948,-56.982,-177.441,6.156,148.349
C06152=1219.968,203.196,-57.006,-177.439,6.158,148.348
C06153=1219.963,203.445,-57.030,-177.436,6.160,148.348
C06154=1219.959,203.694,-57.054,-177.433,6.162,148.347
C06155=1219.954,203.943,-57.077,-177.431,6.163,148.347
C06156=1219.950,204.191,-57.101,-177.428,6.165,148.347
C06157=1219.945,204.440,-57.126,-177.425,6.167,148.346
C06158=1219.941,204.689,-57.150,-177.423,6.168,148.346
C06159=1219.936,204.938,-57.174,-177.420,6.170,148.346
C06160=1219.932,205.186,-57.198,-177.418,6.171,148.345
C06161=1219.926,205.436,-57.222,-177.415,6.173,148.345
C06162=1219.922,205.684,-57.246,-177.412,6.175,148.345
C06163=1219.918,205.932,-57.270,-177.410,6.177,148.344
C06164=1219.914,206.182,-57.294,-177.407,6.179,148.344
C06165=1219.908,206.431,-57.318,-177.404,6.181,148.344
C06166=1219.904,206.679,-57.342,-177.402,6.182,148.343
C06167=1219.900,206.928,-57.366,-177.400,6.184,148.343
C06168=1219.895,207.177,-57.390,-177.397,6.185,148.342
C06169=1219.890,207.425,-57.414,-177.394,6.187,148.342
C06170=1219.886,207.675,-57.439,-177.392,6.189,148.342
C06171=1219.882,207.923,-57.463,-177.389,6.191,148.341
C06172=1219.877,208.172,-57.488,-177.387,6.193,148.341
C06173=1219.872,208.421,-57.511,-177.384,6.195,148.341
C06174=1219.868,208.670,-57.535,-177.382,6.196,148.340
C06175=1219.863,208.919,-57.560,-177.379,6.197,148.340
C06176=1219.858,209.167,-57.584,-177.377,6.199,148.340
C06177=1219.854,209.415,-57.608,-177.374,6.201,148.339
C06178=1219.849,209.664,-57.633,-177.371,6.203,148.339
C06179=1219.845,209.914,-57.657,-177.369,6.205,148.339
C06180=1219.840,210.163,-57.681,-177.366,6.207,148.338
C06181=1219.835,210.411,-57.705,-177.363,6.209,148.338
C06182=1219.831,210.659,-57.729,-177.361,6.210,148.338
C06183=1219.826,210.909,-57.754,-177.358,6.212,148.337
C06184=1219.822,211.179,-57.781,-177.355,6.214,148.337
C06185=1219.817,211.449,-57.807,-177.353,6.216,148.337
C06186=1219.811,211.720,-57.833,-177.350,6.218,148.336
C06187=1219.807,211.991,-57.860,-177.347,6.219,148.336
C06188=1219.802,212.239,-57.884,-177.344,6.221,148.336
C06189=1219.797,212.488,-57.909,-177.342,6.223,148.335
C06190=1219.793,212.736,-57.933,-177.340,6.225,148.335
C06191=1219.788,212.985,-57.958,-177.337,6.227,148.335
C06192=1219.784,213.234,-57.982,-177.334,6.229,148.334
C06193=1219.779,213.483,-58.007,-177.332,6.231,148.334
C06194=1219.775,213.732,-58.031,-177.329,6.233,148.334
C06195=1219.770,213.980,-58.056,-177.326,6.234,148.333
C06196=1219.766,214.229,-58.080,-177.324,6.235,148.333
C06197=1219.761,214.478,-58.105,-177.322,6.237,148.333
C06198=1219.757,214.727,-58.129,-177.319,6.239,148.332
C06199=1219.751,214.975,-58.154,-177.316,6.241,148.332
C06200=1219.748,215.224,-58.179,-177.314,6.243,148.332
C06201=1219.743,215.473,-58.204,-177.311,6.245,148.331
C06202=1219.738,215.721,-58.228,-177.309,6.247,148.331
C06203=1219.734,215.970,-58.253,-177.306,6.248,148.331
C06204=1219.730,216.219,-58.277,-177.303,6.250,148.330
C06205=1219.724,216.468,-58.302,-177.301,6.252,148.330
C06206=1219.721,216.717,-58.326,-177.298,6.254,148.330
C06207=1219.716,216.965,-58.351,-177.295,6.256,148.329
C06208=1219.711,217.214,-58.376,-177.293,6.258,148.329
C06209=1219.707,217.463,-58.400,-177.290,6.260,148.329
C06210=1219.702,217.711,-58.425,-177.288,6.261,148.328
C06211=1219.698,217.961,-58.450,-177.285,6.263,148.328
C06212=1219.693,218.209,-58.475,-177.283,6.264,148.328
C06213=1219.688,218.457,-58.500,-177.280,6.266,148.327
C06214=1219.684,218.706,-58.524,-177.278,6.268,148.327
C06215=1219.679,218.955,-58.549,-177.275,6.270,148.327
C06216=1219.676,219.204,-58.574,-177.273,6.272,148.327
C06217=1219.670,219.452,-58.599,-177.270,6.274,148.326
C06218=1219.665,219.701,-58.623,-177.267,6.276,148.326
C06219=1219.662,219.950,-58.648,-177.265,6.278,148.326
C06220=1219.657,220.198,-58.673,-177.262,6.279,148.325
C06221=1219.652,220.448,-58.698,-177.260,6.281,148.325
C06222=1219.648,220.696,-58.723,-177.257,6.283,148.325
C06223=1219.644,220.945,-58.748,-177.254,6.285,148.324
C06224=1219.638,221.194,-58.773,-177.252,6.287,148.324
C06225=1219.635,221.442,-58.798,-177.249,6.289,148.324
C06226=1219.630,221.691,-58.822,-177.246,6.291,148.323
C06227=1219.625,221.940,-58.847,-177.244,6.292,148.323
C06228=1219.620,222.188,-58.873,-177.241,6.294,148.323
C06229=1219.616,222.437,-58.897,-177.239,6.296,148.323
C06230=1219.612,222.686,-58.923,-177.236,6.298,148.322
C06231=1219.607,222.934,-58.947,-177.234,6.300,148.322
C06232=1219.602,223.183,-58.973,-177.231,6.302,148.322
C06233=1219.598,223.432,-58.997,-177.229,6.304,148.321
C06234=1219.594,223.680,-59.023,-177.226,6.306,148.321
C06235=1219.589,223.929,-59.048,-177.223,6.308,148.321
C06236=1219.584,224.178,-59.073,-177.221,6.309,148.320
C06237=1219.580,224.426,-59.097,-177.219,6.310,148.320
C06238=1219.576,224.675,-59.123,-177.216,6.312,148.320
C06239=1219.571,224.924,-59.148,-177.214,6.314,148.319
C06240=1219.567,225.173,-59.174,-177.211,6.316,148.319
C06241=1219.561,225.421,-59.198,-177.209,6.318,148.319
C06242=1219.558,225.670,-59.223,-177.206,6.320,148.318
C06243=1219.553,225.919,-59.248,-177.203,6.322,148.318
C06244=1219.549,226.167,-59.274,-177.201,6.324,148.318
C06245=1219.544,226.416,-59.300,-177.198,6.326,148.318
C06246=1219.539,226.665,-59.324,-177.195,6.327,148.317
C06247=1219.535,226.914,-59.350,-177.193,6.330,148.317
C06248=1219.530,227.162,-59.375,-177.191,6.332,148.317
C06249=1219.526,227.411,-59.400,-177.188,6.333,148.316
C06250=1219.522,227.659,-59.425,-177.185,6.335,148.316
C06251=1219.517,227.909,-59.450,-177.183,6.337,148.316
C06252=1219.512,228.157,-59.476,-177.180,6.339,148.315
C06253=1219.508,228.405,-59.501,-177.177,6.341,148.315
C06254=1219.503,228.655,-59.526,-177.175,6.343,148.315
C06255=1219.499,228.903,-59.552,-177.173,6.345,148.315
C06256=1219.494,229.152,-59.578,-177.170,6.347,148.314
C06257=1219.490,229.400,-59.603,-177.167,6.349,148.314
C06258=1219.485,229.649,-59.628,-177.165,6.350,148.314
C06259=1219.481,229.898,-59.654,-177.162,6.352,148.313
C06260=1219.476,230.146,-59.679,-177.160,6.354,148.313
C06261=1219.472,230.395,-59.705,-177.157,6.356,148.313
C06262=1219.467,230.644,-59.730,-177.155,6.358,148.313
C06263=1219.462,230.893,-59.755,-177.152,6.360,148.312
C06264=1219.459,231.141,-59.780,-177.150,6.362,148.312
C06265=1219.454,231.389,-59.806,-177.147,6.364,148.312
C06266=1219.450,231.638,-59.832,-177.144,6.366,148.311
C06267=1219.445,231.888,-59.857,-177.142,6.368,148.311
C06268=1219.440,232.136,-59.883,-177.140,6.370,148.311
C06269=1219.436,232.385,-59.908,-177.137,6.372,148.311
C06270=1219.431,232.633,-59.934,-177.134,6.373,148.310
C06271=1219.426,232.881,-59.959,-177.132,6.375,148.310
C06272=1219.422,233.130,-59.985,-177.129,6.377,148.310
C06273=1219.417,233.378,-60.011,-177.127,6.379,148.310
C06274=1219.413,233.627,-60.036,-177.124,6.381,148.309
C06275=1219.409,233.877,-60.061,-177.122,6.383,148.309
C06276=1219.404,234.125,-60.087,-177.119,6.385,148.309
C06277=1219.400,234.374,-60.113,-177.116,6.387,148.308
C06278=1219.395,234.622,-60.138,-177.114,6.389,148.308
C06279=1219.391,234.871,-60.164,-177.112,6.391,148.308
C06280=1219.386,235.119,-60.189,-177.109,6.393,148.308
C06281=1219.382,235.368,-60.215,-177.106,6.395,148.307
C06282=1219.377,235.617,-60.242,-177.104,6.396,148.307
C06283=1219.372,235.865,-60.267,-177.102,6.399,148.307
C06284=1219.368,236.114,-60.293,-177.099,6.400,148.307
C06285=1219.364,236.363,-60.318,-177.096,6.402,148.306
C06286=1219.360,236.612,-60.344,-177.093,6.405,148.306
C06287=1219.355,236.860,-60.370,-177.091,6.407,148.306
C06288=1219.350,237.131,-60.398,-177.088,6.409,148.305
C06289=1219.345,237.402,-60.426,-177.085,6.411,148.305
C06290=1219.340,237.674,-60.454,-177.083,6.413,148.305
C06291=1219.335,237.946,-60.483,-177.080,6.416,148.305
C06292=1219.330,238.194,-60.509,-177.077,6.417,148.304
C06293=1219.326,238.443,-60.534,-177.075,6.419,148.304
C06294=1219.322,238.691,-60.560,-177.072,6.421,148.304
C06295=1219.318,238.940,-60.586,-177.070,6.423,148.303
C06296=1219.313,239.188,-60.613,-177.067,6.425,148.303
C06297=1219.308,239.437,-60.638,-177.065,6.427,148.303
C06298=1219.304,239.686,-60.664,-177.062,6.429,148.303
C06299=1219.300,239.934,-60.690,-177.060,6.431,148.302
C06300=1219.295,240.184,-60.716,-177.057,6.433,148.302
C06301=1219.290,240.431,-60.742,-177.055,6.435,148.302
C06302=1219.286,240.680,-60.768,-177.052,6.437,148.302
C06303=1219.282,240.929,-60.794,-177.050,6.439,148.301
C06304=1219.277,241.178,-60.820,-177.047,6.441,148.301
C06305=1219.273,241.426,-60.847,-177.044,6.443,148.301
C06306=1219.268,241.674,-60.872,-177.042,6.445,148.301
C06307=1219.263,241.923,-60.898,-177.039,6.447,148.300
C06308=1219.259,242.172,-60.924,-177.037,6.449,148.300
C06309=1219.255,242.420,-60.951,-177.034,6.451,148.300
C06310=1219.250,242.669,-60.977,-177.032,6.453,148.300
C06311=1219.246,242.918,-61.003,-177.029,6.455,148.299
C06312=1219.241,243.166,-61.029,-177.027,6.457,148.299
C06313=1219.236,243.415,-61.055,-177.024,6.459,148.299
C06314=1219.232,243.664,-61.081,-177.022,6.461,148.299
C06315=1219.228,243.912,-61.107,-177.019,6.463,148.298
C06316=1219.223,244.161,-61.134,-177.017,6.465,148.298
C06317=1219.219,244.409,-61.160,-177.014,6.467,148.298
C06318=1219.215,244.658,-61.186,-177.012,6.469,148.297
C06319=1219.210,244.906,-61.212,-177.009,6.472,148.297
C06320=1219.206,245.154,-61.238,-177.006,6.474,148.297
C06321=1219.201,245.404,-61.265,-177.004,6.475,148.297
C06322=1219.197,245.652,-61.291,-177.001,6.477,148.296
C06323=1219.193,245.901,-61.317,-176.999,6.479,148.296
C06324=1219.188,246.149,-61.344,-176.996,6.481,148.296
C06325=1219.184,246.398,-61.370,-176.994,6.483,148.296
C06326=1219.179,246.646,-61.397,-176.992,6.485,148.296
C06327=1219.175,246.895,-61.423,-176.989,6.487,148.295
C06328=1219.170,247.144,-61.450,-176.986,6.489,148.295
C06329=1219.165,247.392,-61.475,-176.984,6.491,148.295
C06330=1219.161,247.640,-61.502,-176.982,6.493,148.295
C06331=1219.157,247.889,-61.528,-176.978,6.496,148.294
C06332=1219.152,248.137,-61.555,-176.976,6.498,148.294
C06333=1219.148,248.386,-61.581,-176.974,6.500,148.294
C06334=1219.143,248.635,-61.608,-176.971,6.502,148.294
C06335=1219.139,248.883,-61.634,-176.968,6.504,148.293
C06336=1219.134,249.132,-61.661,-176.966,6.506,148.293
C06337=1219.130,249.380,-61.687,-176.964,6.508,148.293
C06338=1219.125,249.629,-61.713,-176.961,6.510,148.293
C06339=1219.121,249.878,-61.740,-176.958,6.512,148.292
C06340=1219.117,250.126,-61.767,-176.956,6.515,148.292
C06341=1219.112,250.375,-61.793,-176.953,6.516,148.292
C06342=1219.108,250.623,-61.820,-176.950,6.518,148.292
C06343=1219.104,250.872,-61.846,-176.948,6.520,148.292
C06344=1219.099,251.121,-61.873,-176.946,6.522,148.291
C06345=1219.094,251.369,-61.900,-176.943,6.524,148.291
C06346=1219.090,251.617,-61.926,-176.941,6.526,148.291
C06347=1219.086,251.866,-61.953,-176.938,6.528,148.291
C06348=1219.081,252.115,-61.979,-176.935,6.531,148.290
C06349=1219.077,252.363,-62.006,-176.933,6.533,148.290
C06350=1219.072,252.612,-62.033,-176.930,6.535,148.290
C06351=1219.068,252.860,-62.059,-176.928,6.537,148.290
C06352=1219.063,253.109,-62.086,-176.926,6.539,148.290
C06353=1219.059,253.357,-62.113,-176.923,6.541,148.289
C06354=1219.055,253.606,-62.139,-176.920,6.543,148.289
C06355=1219.050,253.854,-62.166,-176.918,6.545,148.289
C06356=1219.045,254.103,-62.193,-176.915,6.548,148.289
C06357=1219.041,254.351,-62.220,-176.913,6.550,148.288
C06358=1219.036,254.600,-62.246,-176.910,6.552,148.288
C06359=1219.032,254.848,-62.273,-176.908,6.554,148.288
C06360=1219.028,255.097,-62.300,-176.906,6.556,148.288
C06361=1219.023,255.345,-62.327,-176.903,6.558,148.287
C06362=1219.019,255.594,-62.354,-176.900,6.560,148.287
C06363=1219.015,255.842,-62.380,-176.898,6.563,148.287
C06364=1219.010,256.090,-62.407,-176.895,6.565,148.287
C06365=1219.006,256.339,-62.435,-176.893,6.566,148.287
C06366=1219.001,256.588,-62.462,-176.890,6.569,148.286
C06367=1218.997,256.836,-62.488,-176.888,6.571,148.286
C06368=1218.993,257.085,-62.515,-176.886,6.573,148.286
C06369=1218.988,257.333,-62.543,-176.882,6.575,148.286
C06370=1218.983,257.582,-62.570,-176.880,6.577,148.285
C06371=1218.979,257.830,-62.597,-176.878,6.579,148.285
C06372=1218.975,258.078,-62.623,-176.875,6.581,148.285
C06373=1218.970,258.327,-62.650,-176.873,6.584,148.285
C06374=1218.966,258.576,-62.678,-176.870,6.585,148.285
C06375=1218.961,258.825,-62.705,-176.867,6.588,148.284
C06376=1218.957,259.073,-62.732,-176.865,6.590,148.284
C06377=1218.953,259.321,-62.758,-176.862,6.592,148.284
C06378=1218.948,259.570,-62.785,-176.860,6.594,148.284
C06379=1218.944,259.818,-62.812,-176.858,6.596,148.284
C06380=1218.939,260.067,-62.839,-176.855,6.598,148.283
C06381=1218.935,260.316,-62.867,-176.852,6.601,148.283
C06382=1218.930,260.564,-62.894,-176.850,6.603,148.283
C06383=1218.926,260.813,-62.920,-176.848,6.605,148.283
C06384=1218.922,261.060,-62.948,-176.845,6.607,148.283
C06385=1218.917,261.309,-62.975,-176.842,6.609,148.282
C06386=1218.913,261.557,-63.002,-176.840,6.611,148.282
C06387=1218.909,261.807,-63.030,-176.837,6.614,148.282
C06388=1218.904,262.055,-63.057,-176.835,6.616,148.282
C06389=1218.900,262.303,-63.084,-176.832,6.618,148.282
C06390=1218.895,262.551,-63.112,-176.830,6.620,148.282
C06391=1218.890,262.800,-63.139,-176.828,6.622,148.281
C06392=1218.886,263.072,-63.168,-176.825,6.625,148.281
C06393=1218.881,263.346,-63.199,-176.822,6.627,148.281
C06394=1218.876,263.618,-63.229,-176.819,6.630,148.281
C06395=1218.871,263.891,-63.258,-176.817,6.632,148.280
C06396=1218.867,264.139,-63.286,-176.814,6.635,148.280
C06397=1218.862,264.388,-63.313,-176.811,6.636,148.280
C06398=1218.858,264.637,-63.341,-176.809,6.639,148.280
C06399=1218.854,264.885,-63.368,-176.807,6.641,148.280
C06400=1218.849,265.133,-63.395,-176.804,6.642,148.279
C06401=1218.844,265.382,-63.422,-176.801,6.645,148.279
C06402=1218.840,265.630,-63.451,-176.799,6.647,148.279
C06403=1218.836,265.879,-63.478,-176.797,6.650,148.279
C06404=1218.831,266.127,-63.505,-176.794,6.651,148.279
C06405=1218.827,266.375,-63.533,-176.791,6.654,148.279
C06406=1218.823,266.624,-63.560,-176.789,6.656,148.278
C06407=1218.818,266.872,-63.588,-176.787,6.659,148.278
C06408=1218.814,267.121,-63.615,-176.784,6.660,148.278
C06409=1218.810,267.369,-63.643,-176.782,6.663,148.278
C06410=1218.805,267.618,-63.670,-176.779,6.665,148.278
C06411=1218.801,267.866,-63.697,-176.777,6.668,148.277
C06412=1218.796,268.114,-63.725,-176.774,6.669,148.277
C06413=1218.792,268.363,-63.752,-176.772,6.672,148.277
C06414=1218.788,268.611,-63.780,-176.769,6.674,148.277
C06415=1218.783,268.860,-63.808,-176.767,6.677,148.277
C06416=1218.779,269.109,-63.836,-176.764,6.678,148.276
C06417=1218.774,269.356,-63.864,-176.762,6.681,148.276
C06418=1218.770,269.605,-63.891,-176.759,6.683,148.276
C06419=1218.766,269.853,-63.919,-176.756,6.686,148.276
C06420=1218.761,270.102,-63.946,-176.754,6.687,148.276
C06421=1218.757,270.350,-63.974,-176.752,6.690,148.276
C06422=1218.752,270.599,-64.002,-176.749,6.691,148.275
C06423=1218.748,270.847,-64.029,-176.746,6.695,148.275
C06424=1218.744,271.095,-64.057,-176.744,6.696,148.275
C06425=1218.739,271.344,-64.085,-176.742,6.699,148.275
C06426=1218.735,271.592,-64.112,-176.739,6.700,148.275
C06427=1218.730,271.841,-64.140,-176.736,6.703,148.275
C06428=1218.726,272.090,-64.168,-176.734,6.705,148.274
C06429=1218.722,272.337,-64.196,-176.732,6.708,148.274
C06430=1218.718,272.587,-64.223,-176.729,6.710,148.274
C06431=1218.713,272.834,-64.251,-176.726,6.712,148.274
C06432=1218.708,273.083,-64.280,-176.724,6.714,148.274
C06433=1218.704,273.331,-64.308,-176.722,6.717,148.274
C06434=1218.700,273.580,-64.335,-176.719,6.720,148.274
C06435=1218.695,273.828,-64.363,-176.716,6.721,148.273
C06436=1218.691,274.077,-64.391,-176.714,6.724,148.273
C06437=1218.687,274.324,-64.419,-176.712,6.726,148.273
C06438=1218.682,274.574,-64.447,-176.709,6.729,148.273
C06439=1218.677,274.822,-64.475,-176.706,6.731,148.273
C06440=1218.674,275.070,-64.503,-176.704,6.733,148.273
C06441=1218.669,275.318,-64.531,-176.702,6.735,148.272
C06442=1218.664,275.566,-64.559,-176.699,6.738,148.272
C06443=1218.660,275.816,-64.587,-176.697,6.740,148.272
C06444=1218.656,276.063,-64.614,-176.694,6.742,148.272
C06445=1218.651,276.312,-64.643,-176.692,6.745,148.272
C06446=1218.647,276.560,-64.671,-176.689,6.747,148.272
C06447=1218.643,276.809,-64.699,-176.687,6.749,148.271
C06448=1218.638,277.057,-64.727,-176.684,6.751,148.271
C06449=1218.634,277.306,-64.756,-176.682,6.754,148.271
C06450=1218.630,277.553,-64.783,-176.679,6.756,148.271
C06451=1218.626,277.802,-64.812,-176.677,6.758,148.271
C06452=1218.621,278.050,-64.840,-176.674,6.761,148.271
C06453=1218.617,278.299,-64.867,-176.672,6.763,148.270
C06454=1218.612,278.548,-64.896,-176.669,6.765,148.270
C06455=1218.608,278.796,-64.924,-176.667,6.767,148.270
C06456=1218.603,279.044,-64.952,-176.664,6.770,148.270
C06457=1218.599,279.293,-64.980,-176.662,6.772,148.270
C06458=1218.594,279.541,-65.009,-176.659,6.774,148.270
C06459=1218.591,279.790,-65.037,-176.657,6.777,148.270
C06460=1218.586,280.038,-65.065,-176.655,6.779,148.270
C06461=1218.582,280.286,-65.093,-176.652,6.781,148.269
C06462=1218.578,280.534,-65.122,-176.649,6.784,148.269
C06463=1218.573,280.783,-65.151,-176.647,6.786,148.269
C06464=1218.569,281.030,-65.178,-176.645,6.788,148.269
C06465=1218.564,281.279,-65.207,-176.643,6.790,148.269
C06466=1218.560,281.527,-65.235,-176.639,6.793,148.269
C06467=1218.556,281.776,-65.264,-176.637,6.795,148.269
C06468=1218.551,282.024,-65.291,-176.635,6.798,148.268
C06469=1218.547,282.273,-65.320,-176.632,6.800,148.268
C06470=1218.543,282.521,-65.348,-176.630,6.802,148.268
C06471=1218.538,282.769,-65.377,-176.628,6.805,148.268
C06472=1218.534,283.018,-65.406,-176.625,6.807,148.268
C06473=1218.529,283.266,-65.434,-176.622,6.810,148.268
C06474=1218.525,283.515,-65.463,-176.620,6.812,148.268
C06475=1218.520,283.763,-65.490,-176.617,6.815,148.267
C06476=1218.516,284.011,-65.520,-176.615,6.817,148.267
C06477=1218.513,284.259,-65.548,-176.613,6.819,148.267
C06478=1218.507,284.508,-65.576,-176.610,6.822,148.267
C06479=1218.503,284.756,-65.605,-176.608,6.824,148.267
C06480=1218.499,285.004,-65.634,-176.606,6.826,148.267
C06481=1218.494,285.253,-65.662,-176.602,6.829,148.267
C06482=1218.491,285.501,-65.690,-176.600,6.831,148.267
C06483=1218.486,285.749,-65.719,-176.598,6.833,148.267
C06484=1218.481,285.998,-65.748,-176.595,6.836,148.267
C06485=1218.478,286.246,-65.776,-176.593,6.838,148.266
C06486=1218.473,286.494,-65.805,-176.591,6.840,148.266
C06487=1218.468,286.743,-65.834,-176.588,6.843,148.266
C06488=1218.465,286.991,-65.862,-176.585,6.845,148.266
C06489=1218.460,287.239,-65.891,-176.583,6.847,148.266
C06490=1218.455,287.488,-65.920,-176.581,6.851,148.266
C06491=1218.451,287.736,-65.948,-176.578,6.852,148.266
C06492=1218.447,287.984,-65.977,-176.576,6.855,148.265
C06493=1218.442,288.233,-66.006,-176.573,6.858,148.265
C06494=1218.437,288.481,-66.035,-176.571,6.860,148.265
C06495=1218.434,288.729,-66.063,-176.569,6.862,148.265
C06496=1218.429,289.003,-66.095,-176.566,6.865,148.265
C06497=1218.424,289.278,-66.127,-176.563,6.868,148.265
C06498=1218.420,289.551,-66.159,-176.560,6.871,148.265
C06499=1218.415,289.826,-66.191,-176.558,6.873,148.265
C06500=1218.410,290.075,-66.219,-176.555,6.876,148.265
C06501=1218.406,290.322,-66.248,-176.553,6.878,148.264
C06502=1218.401,290.571,-66.277,-176.551,6.880,148.264
C06503=1218.398,290.819,-66.306,-176.548,6.883,148.264
C06504=1218.393,291.067,-66.335,-176.546,6.885,148.264
C06505=1218.388,291.315,-66.364,-176.543,6.887,148.264
C06506=1218.384,291.564,-66.393,-176.540,6.890,148.264
C06507=1218.380,291.813,-66.422,-176.538,6.892,148.264
C06508=1218.376,292.060,-66.451,-176.536,6.895,148.264
C06509=1218.372,292.308,-66.480,-176.533,6.897,148.264
C06510=1218.367,292.557,-66.509,-176.531,6.899,148.264
C06511=1218.363,292.805,-66.538,-176.528,6.902,148.264
C06512=1218.358,293.053,-66.567,-176.526,6.905,148.263
C06513=1218.354,293.302,-66.596,-176.524,6.907,148.263
C06514=1218.349,293.550,-66.626,-176.521,6.910,148.263
C06515=1218.346,293.799,-66.654,-176.519,6.912,148.263
C06516=1218.342,294.047,-66.683,-176.516,6.915,148.263
C06517=1218.337,294.294,-66.712,-176.514,6.917,148.263
C06518=1218.333,294.543,-66.742,-176.512,6.919,148.263
C06519=1218.328,294.792,-66.770,-176.509,6.922,148.263
C06520=1218.324,295.040,-66.800,-176.507,6.924,148.263
C06521=1218.319,295.287,-66.829,-176.505,6.926,148.263
C06522=1218.315,295.536,-66.858,-176.502,6.929,148.263
C06523=1218.310,295.785,-66.887,-176.500,6.932,148.263
C06524=1218.306,296.033,-66.917,-176.497,6.935,148.263
C06525=1218.302,296.281,-66.946,-176.494,6.937,148.262
C06526=1218.298,296.529,-66.975,-176.492,6.939,148.262
C06527=1218.293,296.777,-67.005,-176.490,6.942,148.262
C06528=1218.289,297.026,-67.033,-176.488,6.944,148.262
C06529=1218.285,297.274,-67.062,-176.485,6.947,148.262
C06530=1218.281,297.522,-67.092,-176.483,6.949,148.262
C06531=1218.277,297.770,-67.121,-176.481,6.951,148.262
C06532=1218.273,298.019,-67.151,-176.478,6.954,148.262
C06533=1218.268,298.267,-67.180,-176.475,6.956,148.262
C06534=1218.264,298.514,-67.209,-176.473,6.959,148.262
C06535=1218.259,298.763,-67.239,-176.471,6.962,148.262
C06536=1218.254,299.012,-67.268,-176.468,6.964,148.262
C06537=1218.250,299.260,-67.297,-176.466,6.967,148.262
C06538=1218.246,299.508,-67.327,-176.464,6.969,148.261
C06539=1218.242,299.757,-67.356,-176.461,6.972,148.261
C06540=1218.238,300.005,-67.386,-176.459,6.974,148.261
C06541=1218.233,300.253,-67.415,-176.456,6.976,148.261
C06542=1218.229,300.501,-67.444,-176.454,6.979,148.261
C06543=1218.224,300.749,-67.474,-176.452,6.982,148.261
C06544=1218.220,300.997,-67.503,-176.449,6.985,148.261
C06545=1218.216,301.246,-67.533,-176.447,6.987,148.261
C06546=1218.212,301.494,-67.562,-176.445,6.989,148.261
C06547=1218.208,301.742,-67.591,-176.442,6.992,148.261
C06548=1218.203,301.990,-67.622,-176.440,6.994,148.261
C06549=1218.199,302.238,-67.652,-176.437,6.997,148.261
C06550=1218.195,302.487,-67.681,-176.435,7.000,148.261
C06551=1218.190,302.735,-67.711,-176.433,7.002,148.261
C06552=1218.186,302.983,-67.740,-176.430,7.005,148.261
C06553=1218.182,303.231,-67.770,-176.428,7.007,148.261
C06554=1218.177,303.480,-67.800,-176.425,7.010,148.261
C06555=1218.172,303.728,-67.829,-176.423,7.012,148.261
C06556=1218.168,303.976,-67.858,-176.420,7.015,148.260
C06557=1218.164,304.223,-67.888,-176.418,7.017,148.260
C06558=1218.160,304.472,-67.918,-176.416,7.019,148.260
C06559=1218.155,304.720,-67.948,-176.413,7.022,148.260
C06560=1218.151,304.969,-67.977,-176.411,7.025,148.260
C06561=1218.147,305.217,-68.007,-176.409,7.028,148.260
C06562=1218.143,305.464,-68.037,-176.406,7.030,148.260
C06563=1218.138,305.713,-68.067,-176.404,7.033,148.260
C06564=1218.134,305.961,-68.096,-176.402,7.035,148.260
C06565=1218.130,306.210,-68.126,-176.400,7.037,148.260
C06566=1218.126,306.457,-68.156,-176.397,7.040,148.260
C06567=1218.121,306.706,-68.186,-176.395,7.043,148.260
C06568=1218.117,306.954,-68.215,-176.392,7.046,148.260
C06569=1218.113,307.202,-68.246,-176.390,7.048,148.260
C06570=1218.109,307.450,-68.275,-176.387,7.051,148.260
C06571=1218.104,307.699,-68.305,-176.385,7.053,148.260
C06572=1218.100,307.946,-68.335,-176.383,7.055,148.260
C06573=1218.096,308.195,-68.365,-176.381,7.059,148.260
C06574=1218.091,308.443,-68.395,-176.379,7.061,148.260
C06575=1218.087,308.691,-68.425,-176.376,7.064,148.260
C06576=1218.083,308.939,-68.454,-176.374,7.066,148.260
C06577=1218.079,309.188,-68.486,-176.371,7.069,148.260
C06578=1218.075,309.436,-68.515,-176.369,7.071,148.260
C06579=1218.070,309.685,-68.545,-176.367,7.074,148.260
C06580=1218.066,309.932,-68.575,-176.364,7.077,148.260
C06581=1218.062,310.180,-68.605,-176.362,7.079,148.260
C06582=1218.057,310.428,-68.635,-176.360,7.082,148.260
C06583=1218.053,310.677,-68.665,-176.357,7.084,148.260
C06584=1218.049,310.924,-68.695,-176.355,7.087,148.260
C06585=1218.044,311.173,-68.725,-176.353,7.089,148.260
C06586=1218.040,311.421,-68.755,-176.350,7.092,148.260
C06587=1218.035,311.669,-68.785,-176.348,7.095,148.260
C06588=1218.031,311.917,-68.816,-176.346,7.098,148.260
C06589=1218.027,312.166,-68.846,-176.344,7.100,148.260
C06590=1218.023,312.414,-68.876,-176.342,7.102,148.260
C06591=1218.019,312.662,-68.907,-176.339,7.105,148.260
C06592=1218.014,312.910,-68.936,-176.337,7.108,148.260
C06593=1218.010,313.158,-68.966,-176.334,7.111,148.260
C06594=1218.006,313.406,-68.997,-176.332,7.113,148.260
C06595=1218.002,313.654,-69.027,-176.330,7.116,148.260
C06596=1217.997,313.902,-69.057,-176.328,7.118,148.260
C06597=1217.993,314.151,-69.087,-176.325,7.122,148.260
C06598=1217.989,314.399,-69.118,-176.323,7.124,148.260
C06599=1217.985,314.646,-69.148,-176.321,7.126,148.260
C06600=1217.980,314.923,-69.182,-176.318,7.129,148.260
C06601=1217.975,315.199,-69.216,-176.315,7.132,148.260
C06602=1217.971,315.475,-69.249,-176.313,7.135,148.260
C06603=1217.966,315.750,-69.283,-176.310,7.138,148.260
C06604=1217.961,315.999,-69.313,-176.308,7.141,148.260
C06605=1217.957,316.247,-69.344,-176.306,7.144,148.260
C06606=1217.953,316.495,-69.374,-176.304,7.146,148.260
C06607=1217.949,316.742,-69.404,-176.301,7.149,148.260
C06608=1217.944,316.992,-69.435,-176.299,7.151,148.260
C06609=1217.940,317.239,-69.466,-176.297,7.155,148.260
C06610=1217.936,317.487,-69.496,-176.295,7.157,148.260
C06611=1217.931,317.735,-69.527,-176.292,7.159,148.260
C06612=1217.927,317.983,-69.557,-176.290,7.162,148.260
C06613=1217.923,318.231,-69.588,-176.288,7.165,148.260
C06614=1217.918,318.480,-69.618,-176.286,7.168,148.260
C06615=1217.915,318.728,-69.648,-176.283,7.170,148.260
C06616=1217.910,318.976,-69.679,-176.281,7.173,148.260
C06617=1217.906,319.224,-69.710,-176.279,7.175,148.260
C06618=1217.902,319.472,-69.740,-176.276,7.178,148.260
C06619=1217.898,319.720,-69.771,-176.274,7.181,148.260
C06620=1217.893,319.968,-69.802,-176.272,7.184,148.260
C06621=1217.890,320.216,-69.832,-176.270,7.186,148.260
C06622=1217.885,320.464,-69.863,-176.267,7.189,148.260
C06623=1217.880,320.712,-69.894,-176.265,7.191,148.260
C06624=1217.877,320.960,-69.924,-176.264,7.194,148.260
C06625=1217.873,321.208,-69.955,-176.261,7.197,148.260
C06626=1217.868,321.457,-69.985,-176.259,7.199,148.260
C06627=1217.863,321.705,-70.016,-176.256,7.202,148.260
C06628=1217.860,321.953,-70.047,-176.255,7.205,148.260
C06629=1217.855,322.201,-70.078,-176.252,7.208,148.260
C06630=1217.851,322.449,-70.109,-176.250,7.210,148.260
C06631=1217.846,322.696,-70.139,-176.248,7.213,148.261
C06632=1217.843,322.945,-70.170,-176.245,7.216,148.261
C06633=1217.838,323.193,-70.201,-176.243,7.219,148.261
C06634=1217.834,323.441,-70.231,-176.241,7.221,148.261
C06635=1217.830,323.689,-70.263,-176.238,7.224,148.261
C06636=1217.826,323.937,-70.293,-176.236,7.226,148.261
C06637=1217.821,324.185,-70.324,-176.235,7.229,148.261
C06638=1217.817,324.434,-70.355,-176.232,7.232,148.261
C06639=1217.813,324.682,-70.385,-176.230,7.235,148.261
C06640=1217.808,324.929,-70.417,-176.228,7.238,148.261
C06641=1217.805,325.177,-70.447,-176.226,7.240,148.261
C06642=1217.800,325.425,-70.478,-176.223,7.243,148.261
C06643=1217.796,325.673,-70.509,-176.221,7.245,148.261
C06644=1217.792,325.922,-70.540,-176.219,7.248,148.261
C06645=1217.787,326.169,-70.572,-176.217,7.251,148.261
C06646=1217.783,326.418,-70.603,-176.214,7.254,148.261
C06647=1217.779,326.666,-70.633,-176.213,7.257,148.262
C06648=1217.775,326.913,-70.664,-176.210,7.260,148.262
C06649=1217.771,327.162,-70.695,-176.208,7.262,148.262
C06650=1217.767,327.409,-70.726,-176.206,7.264,148.262
C06651=1217.762,327.657,-70.757,-176.204,7.267,148.262
C06652=1217.758,327.906,-70.788,-176.202,7.270,148.262
C06653=1217.754,328.153,-70.820,-176.199,7.273,148.262
C06654=1217.750,328.402,-70.851,-176.198,7.275,148.262
C06655=1217.745,328.650,-70.881,-176.195,7.278,148.262
C06656=1217.741,328.897,-70.913,-176.193,7.281,148.262
C06657=1217.737,329.146,-70.944,-176.191,7.284,148.262
C06658=1217.732,329.394,-70.975,-176.189,7.287,148.262
C06659=1217.728,329.642,-71.007,-176.186,7.290,148.262
C06660=1217.724,329.890,-71.037,-176.185,7.292,148.263
C06661=1217.720,330.139,-71.069,-176.182,7.295,148.263
C06662=1217.715,330.386,-71.100,-176.180,7.298,148.263
C06663=1217.711,330.634,-71.131,-176.178,7.301,148.263
C06664=1217.707,330.882,-71.163,-176.176,7.303,148.263
C06665=1217.703,331.130,-71.193,-176.174,7.306,148.263
C06666=1217.699,331.378,-71.225,-176.172,7.309,148.263
C06667=1217.694,331.626,-71.256,-176.170,7.311,148.263
C06668=1217.690,331.874,-71.288,-176.168,7.314,148.263
C06669=1217.686,332.122,-71.319,-176.165,7.317,148.263
C06670=1217.682,332.371,-71.350,-176.163,7.320,148.263
C06671=1217.678,332.618,-71.381,-176.162,7.323,148.264
C06672=1217.674,332.866,-71.413,-176.159,7.326,148.264
C06673=1217.669,333.114,-71.444,-176.157,7.328,148.264
C06674=1217.666,333.362,-71.476,-176.155,7.331,148.264
C06675=1217.661,333.610,-71.507,-176.153,7.334,148.264
C06676=1217.657,333.858,-71.538,-176.151,7.336,148.264
C06677=1217.653,334.106,-71.569,-176.149,7.339,148.264
C06678=1217.649,334.354,-71.601,-176.147,7.342,148.264
C06679=1217.644,334.602,-71.632,-176.144,7.345,148.264
C06680=1217.640,334.850,-71.664,-176.143,7.347,148.265
C06681=1217.636,335.098,-71.696,-176.141,7.351,148.265
C06682=1217.632,335.346,-71.727,-176.138,7.353,148.265
C06683=1217.627,335.594,-71.758,-176.136,7.356,148.265
C06684=1217.624,335.842,-71.790,-176.135,7.359,148.265
C06685=1217.619,336.090,-71.821,-176.132,7.362,148.265
C06686=1217.614,336.338,-71.853,-176.130,7.364,148.265
C06687=1217.610,336.585,-71.885,-176.129,7.367,148.265
C06688=1217.606,336.834,-71.916,-176.126,7.370,148.266
C06689=1217.602,337.081,-71.947,-176.124,7.372,148.266
C06690=1217.598,337.329,-71.979,-176.122,7.376,148.266
C06691=1217.594,337.577,-72.011,-176.120,7.378,148.266
C06692=1217.589,337.826,-72.042,-176.118,7.381,148.266
C06693=1217.585,338.074,-72.074,-176.116,7.384,148.266
C06694=1217.581,338.321,-72.106,-176.114,7.387,148.266
C06695=1217.577,338.569,-72.138,-176.112,7.389,148.266
C06696=1217.573,338.818,-72.169,-176.110,7.393,148.267
C06697=1217.568,339.065,-72.201,-176.108,7.395,148.267
C06698=1217.565,339.313,-72.233,-176.106,7.398,148.267
C06699=1217.560,339.561,-72.264,-176.104,7.401,148.267
C06700=1217.556,339.809,-72.297,-176.102,7.403,148.267
C06701=1217.552,340.057,-72.328,-176.100,7.407,148.267
C06702=1217.548,340.305,-72.359,-176.098,7.409,148.267
C06703=1217.544,340.553,-72.391,-176.096,7.412,148.268
C06704=1217.539,340.831,-72.427,-176.094,7.415,148.268
C06705=1217.534,341.109,-72.463,-176.092,7.418,148.268
C06706=1217.529,341.387,-72.498,-176.089,7.421,148.268
C06707=1217.525,341.665,-72.534,-176.087,7.425,148.268
C06708=1217.521,341.913,-72.566,-176.085,7.427,148.268
C06709=1217.516,342.160,-72.598,-176.083,7.431,148.269
C06710=1217.512,342.408,-72.630,-176.082,7.433,148.269
C06711=1217.508,342.657,-72.662,-176.079,7.436,148.269
C06712=1217.504,342.904,-72.694,-176.077,7.439,148.269
C06713=1217.500,343.152,-72.725,-176.075,7.442,148.269
C06714=1217.495,343.400,-72.758,-176.073,7.444,148.269
C06715=1217.491,343.648,-72.789,-176.072,7.447,148.270
C06716=1217.487,343.896,-72.821,-176.070,7.450,148.270
C06717=1217.482,344.143,-72.853,-176.068,7.453,148.270
C06718=1217.479,344.391,-72.885,-176.066,7.456,148.270
C06719=1217.474,344.640,-72.918,-176.064,7.459,148.270
C06720=1217.470,344.887,-72.949,-176.061,7.462,148.270
C06721=1217.466,345.135,-72.981,-176.060,7.464,148.271
C06722=1217.462,345.383,-73.013,-176.058,7.467,148.271
C06723=1217.458,345.631,-73.045,-176.056,7.470,148.271
C06724=1217.453,345.879,-73.077,-176.054,7.473,148.271
C06725=1217.449,346.127,-73.109,-176.052,7.476,148.271
C06726=1217.445,346.375,-73.142,-176.050,7.479,148.272
C06727=1217.441,346.622,-73.174,-176.048,7.482,148.272
C06728=1217.436,346.871,-73.206,-176.047,7.484,148.272
C06729=1217.433,347.119,-73.238,-176.045,7.487,148.272
C06730=1217.428,347.367,-73.270,-176.043,7.490,148.272
C06731=1217.424,347.614,-73.302,-176.041,7.493,148.273
C06732=1217.420,347.862,-73.335,-176.039,7.496,148.273
C06733=1217.416,348.110,-73.367,-176.037,7.499,148.273
C06734=1217.411,348.358,-73.399,-176.036,7.501,148.273
C06735=1217.407,348.606,-73.431,-176.033,7.505,148.273
C06736=1217.403,348.854,-73.463,-176.032,7.507,148.274
C06737=1217.399,349.102,-73.496,-176.030,7.511,148.274
C06738=1217.394,349.349,-73.528,-176.028,7.513,148.274
C06739=1217.391,349.597,-73.560,-176.026,7.516,148.274
C06740=1217.387,349.845,-73.593,-176.024,7.519,148.274
C06741=1217.383,350.093,-73.625,-176.023,7.521,148.275
C06742=1217.378,350.341,-73.657,-176.020,7.525,148.275
C06743=1217.373,350.589,-73.689,-176.019,7.527,148.275
C06744=1217.370,350.836,-73.722,-176.017,7.530,148.275
C06745=1217.366,351.085,-73.754,-176.015,7.533,148.275
C06746=1217.362,351.333,-73.786,-176.014,7.536,148.276
C06747=1217.358,351.581,-73.819,-176.012,7.539,148.276
C06748=1217.353,351.828,-73.851,-176.010,7.542,148.276
C06749=1217.349,352.076,-73.884,-176.008,7.544,148.276
C06750=1217.345,352.324,-73.916,-176.006,7.548,148.277
C06751=1217.341,352.572,-73.948,-176.004,7.550,148.277
C06752=1217.337,352.820,-73.981,-176.003,7.553,148.277
C06753=1217.332,353.067,-74.013,-176.001,7.556,148.277
C06754=1217.329,353.315,-74.046,-175.999,7.559,148.278
C06755=1217.324,353.563,-74.078,-175.997,7.562,148.278
C06756=1217.320,353.811,-74.111,-175.995,7.565,148.278
C06757=1217.316,354.059,-74.143,-175.994,7.567,148.278
C06758=1217.312,354.307,-74.176,-175.992,7.571,148.279
C06759=1217.307,354.554,-74.209,-175.990,7.574,148.279
C06760=1217.303,354.802,-74.241,-175.989,7.576,148.279
C06761=1217.299,355.050,-74.274,-175.987,7.579,148.279
C06762=1217.295,355.298,-74.306,-175.985,7.582,148.279
C06763=1217.291,355.546,-74.339,-175.984,7.585,148.280
C06764=1217.287,355.794,-74.372,-175.982,7.588,148.280
C06765=1217.283,356.042,-74.404,-175.980,7.591,148.280
C06766=1217.278,356.289,-74.437,-175.978,7.593,148.280
C06767=1217.274,356.537,-74.469,-175.977,7.597,148.281
C06768=1217.270,356.785,-74.502,-175.975,7.599,148.281
C06769=1217.266,357.033,-74.535,-175.973,7.603,148.281
C06770=1217.262,357.281,-74.568,-175.971,7.605,148.282
C06771=1217.258,357.528,-74.600,-175.970,7.608,148.282
C06772=1217.254,357.777,-74.633,-175.968,7.611,148.282
C06773=1217.250,358.024,-74.666,-175.966,7.614,148.282
C06774=1217.245,358.272,-74.699,-175.965,7.617,148.283
C06775=1217.241,358.519,-74.730,-175.963,7.620,148.283
C06776=1217.237,358.767,-74.764,-175.961,7.623,148.283
C06777=1217.233,359.015,-74.797,-175.960,7.625,148.284
C06778=1217.228,359.263,-74.829,-175.958,7.629,148.284
C06779=1217.224,359.511,-74.862,-175.956,7.631,148.284
C06780=1217.221,359.758,-74.895,-175.955,7.634,148.284
C06781=1217.216,360.007,-74.927,-175.953,7.637,148.285
C06782=1217.212,360.254,-74.961,-175.951,7.640,148.285
C06783=1217.208,360.502,-74.994,-175.950,7.643,148.285
C06784=1217.204,360.750,-75.027,-175.949,7.646,148.286
C06785=1217.200,360.998,-75.059,-175.946,7.649,148.286
C06786=1217.196,361.246,-75.092,-175.945,7.651,148.286
C06787=1217.192,361.493,-75.125,-175.944,7.654,148.286
C06788=1217.188,361.741,-75.158,-175.941,7.658,148.287
C06789=1217.183,361.989,-75.191,-175.940,7.660,148.287
C06790=1217.179,362.237,-75.224,-175.939,7.663,148.287
C06791=1217.175,362.485,-75.257,-175.937,7.666,148.288
C06792=1217.171,362.733,-75.290,-175.935,7.669,148.288
C06793=1217.167,362.980,-75.323,-175.934,7.672,148.288
C06794=1217.164,363.228,-75.356,-175.932,7.675,148.288
C06795=1217.159,363.476,-75.388,-175.931,7.678,148.289
C06796=1217.155,363.724,-75.421,-175.929,7.681,148.289
C06797=1217.151,363.972,-75.455,-175.928,7.684,148.289
C06798=1217.147,364.219,-75.488,-175.926,7.686,148.290
C06799=1217.143,364.467,-75.521,-175.924,7.690,148.290
C06800=1217.138,364.715,-75.554,-175.923,7.693,148.290
C06801=1217.134,364.962,-75.587,-175.922,7.695,148.291
C06802=1217.130,365.210,-75.620,-175.920,7.698,148.291
C06803=1217.126,365.458,-75.653,-175.918,7.701,148.291
C06804=1217.122,365.706,-75.687,-175.917,7.704,148.292
C06805=1217.118,365.953,-75.720,-175.916,7.707,148.292
C06806=1217.114,366.201,-75.753,-175.914,7.709,148.292
C06807=1217.109,366.449,-75.786,-175.913,7.712,148.293
C06808=1217.105,366.729,-75.823,-175.911,7.716,148.293
C06809=1217.100,367.009,-75.860,-175.909,7.719,148.293
C06810=1217.096,367.289,-75.898,-175.908,7.722,148.294
C06811=1217.091,367.569,-75.935,-175.906,7.726,148.294
C06812=1217.087,367.817,-75.968,-175.905,7.728,148.295
C06813=1217.083,368.065,-76.001,-175.903,7.731,148.295
C06814=1217.079,368.312,-76.035,-175.902,7.734,148.295
C06815=1217.075,368.559,-76.069,-175.900,7.737,148.296
C06816=1217.071,368.807,-76.102,-175.899,7.740,148.296
C06817=1217.067,369.055,-76.135,-175.898,7.743,148.296
C06818=1217.062,369.303,-76.169,-175.896,7.746,148.297
C06819=1217.058,369.551,-76.202,-175.895,7.748,148.297
C06820=1217.053,369.798,-76.235,-175.894,7.751,148.297
C06821=1217.049,370.046,-76.268,-175.892,7.754,148.297
C06822=1217.046,370.295,-76.302,-175.891,7.757,148.298
C06823=1217.042,370.542,-76.335,-175.890,7.760,148.298
C06824=1217.038,370.789,-76.369,-175.888,7.763,148.299
C06825=1217.034,371.037,-76.402,-175.887,7.766,148.299
C06826=1217.029,371.285,-76.435,-175.885,7.768,148.299
C06827=1217.025,371.533,-76.468,-175.884,7.771,148.300
C06828=1217.020,371.781,-76.502,-175.883,7.774,148.300
C06829=1217.016,372.028,-76.535,-175.882,7.777,148.300
C06830=1217.012,372.275,-76.569,-175.881,7.780,148.301
C06831=1217.008,372.523,-76.602,-175.879,7.783,148.301
C06832=1217.005,372.772,-76.636,-175.878,7.786,148.302
C06833=1217.001,373.019,-76.669,-175.876,7.789,148.302
C06834=1216.997,373.266,-76.703,-175.875,7.791,148.302
C06835=1216.992,373.514,-76.736,-175.874,7.794,148.303
C06836=1216.988,373.762,-76.769,-175.873,7.797,148.303
C06837=1216.984,374.010,-76.803,-175.871,7.800,148.303
C06838=1216.980,374.257,-76.836,-175.870,7.803,148.304
C06839=1216.976,374.505,-76.870,-175.869,7.806,148.304
C06840=1216.972,374.753,-76.903,-175.868,7.808,148.305
C06841=1216.968,375.001,-76.938,-175.867,7.811,148.305
C06842=1216.963,375.248,-76.971,-175.865,7.814,148.305
C06843=1216.959,375.496,-77.004,-175.864,7.817,148.306
C06844=1216.955,375.744,-77.037,-175.863,7.820,148.306
C06845=1216.951,375.991,-77.071,-175.862,7.822,148.307
C06846=1216.947,376.240,-77.105,-175.861,7.825,148.307
C06847=1216.943,376.487,-77.139,-175.860,7.828,148.307
C06848=1216.939,376.735,-77.172,-175.858,7.831,148.308
C06849=1216.935,376.982,-77.205,-175.857,7.834,148.308
C06850=1216.930,377.230,-77.240,-175.856,7.837,148.309
C06851=1216.927,377.478,-77.273,-175.855,7.839,148.309
C06852=1216.923,377.726,-77.306,-175.854,7.842,148.309
C06853=1216.919,377.973,-77.340,-175.852,7.845,148.310
C06854=1216.914,378.221,-77.374,-175.851,7.848,148.310
C06855=1216.910,378.468,-77.408,-175.850,7.851,148.311
C06856=1216.906,378.716,-77.441,-175.849,7.853,148.311
C06857=1216.903,378.964,-77.475,-175.848,7.855,148.311
C06858=1216.898,379.212,-77.509,-175.847,7.859,148.312
C06859=1216.894,379.459,-77.542,-175.846,7.861,148.312
C06860=1216.890,379.706,-77.576,-175.845,7.864,148.313
C06861=1216.886,379.955,-77.610,-175.844,7.867,148.313
C06862=1216.882,380.202,-77.644,-175.843,7.870,148.313
C06863=1216.878,380.450,-77.677,-175.842,7.873,148.314
C06864=1216.873,380.697,-77.712,-175.840,7.875,148.314
C06865=1216.869,380.945,-77.745,-175.840,7.879,148.315
C06866=1216.866,381.193,-77.779,-175.839,7.881,148.315
C06867=1216.861,381.441,-77.813,-175.838,7.883,148.316
C06868=1216.857,381.688,-77.847,-175.837,7.886,148.316
C06869=1216.853,381.936,-77.880,-175.835,7.889,148.316
C06870=1216.849,382.184,-77.915,-175.834,7.892,148.317
C06871=1216.845,382.431,-77.949,-175.833,7.895,148.317
C06872=1216.841,382.679,-77.982,-175.832,7.898,148.318
C06873=1216.836,382.926,-78.016,-175.832,7.900,148.318
C06874=1216.833,383.175,-78.050,-175.830,7.902,148.319
C06875=1216.829,383.422,-78.084,-175.830,7.906,148.319
C06876=1216.824,383.670,-78.117,-175.829,7.908,148.320
C06877=1216.820,383.917,-78.151,-175.827,7.911,148.320
C06878=1216.816,384.165,-78.186,-175.827,7.913,148.320
C06879=1216.812,384.413,-78.219,-175.826,7.916,148.321
C06880=1216.808,384.660,-78.253,-175.825,7.919,148.321
C06881=1216.804,384.907,-78.288,-175.824,7.922,148.322
C06882=1216.800,385.156,-78.321,-175.823,7.924,148.322
C06883=1216.796,385.403,-78.355,-175.822,7.927,148.323
C06884=1216.792,385.650,-78.389,-175.821,7.930,148.323
C06885=1216.787,385.898,-78.423,-175.820,7.933,148.323
C06886=1216.784,386.146,-78.457,-175.820,7.935,148.324
C06887=1216.780,386.393,-78.491,-175.818,7.938,148.324
C06888=1216.775,386.641,-78.525,-175.817,7.941,148.325
C06889=1216.772,386.889,-78.559,-175.816,7.943,148.325
C06890=1216.767,387.137,-78.594,-175.816,7.946,148.326
C06891=1216.763,387.384,-78.627,-175.815,7.948,148.326
C06892=1216.759,387.632,-78.662,-175.813,7.951,148.326
C06893=1216.755,387.879,-78.696,-175.813,7.954,148.327
C06894=1216.751,388.127,-78.730,-175.812,7.956,148.327
C06895=1216.747,388.375,-78.763,-175.811,7.960,148.328
C06896=1216.743,388.623,-78.798,-175.811,7.961,148.328
C06897=1216.739,388.870,-78.832,-175.810,7.964,148.329
C06898=1216.734,389.117,-78.866,-175.809,7.967,148.329
C06899=1216.731,389.366,-78.900,-175.808,7.969,148.330
C06900=1216.727,389.613,-78.934,-175.807,7.972,148.330
C06901=1216.722,389.860,-78.968,-175.806,7.975,148.331
C06902=1216.719,390.108,-79.002,-175.806,7.977,148.331
C06903=1216.715,390.355,-79.037,-175.804,7.980,148.331
C06904=1216.710,390.604,-79.071,-175.804,7.982,148.332
C06905=1216.706,390.851,-79.105,-175.803,7.985,148.332
C06906=1216.702,391.099,-79.139,-175.802,7.988,148.333
C06907=1216.698,391.346,-79.173,-175.802,7.990,148.333
C06908=1216.694,391.594,-79.208,-175.801,7.993,148.334
C06909=1216.690,391.841,-79.242,-175.800,7.995,148.334
C06910=1216.686,392.090,-79.276,-175.799,7.998,148.335
C06911=1216.682,392.337,-79.310,-175.799,8.000,148.335
C06912=1216.677,392.619,-79.349,-175.798,8.003,148.336
C06913=1216.672,392.901,-79.388,-175.797,8.006,148.336
C06914=1216.669,393.183,-79.427,-175.796,8.009,148.337
C06915=1216.663,393.465,-79.466,-175.795,8.012,148.337
C06916=1216.659,393.712,-79.500,-175.794,8.015,148.338
C06917=1216.656,393.960,-79.535,-175.794,8.017,148.338
C06918=1216.651,394.208,-79.569,-175.793,8.020,148.339
C06919=1216.647,394.455,-79.603,-175.792,8.022,148.339
C06920=1216.643,394.703,-79.638,-175.791,8.026,148.340
C06921=1216.639,394.950,-79.672,-175.791,8.028,148.340
C06922=1216.635,395.198,-79.706,-175.790,8.031,148.341
C06923=1216.632,395.445,-79.741,-175.789,8.033,148.341
C06924=1216.627,395.693,-79.775,-175.789,8.035,148.341
C06925=1216.623,395.941,-79.810,-175.788,8.038,148.342
C06926=1216.619,396.188,-79.844,-175.787,8.040,148.342
C06927=1216.615,396.435,-79.878,-175.787,8.043,148.343
C06928=1216.611,396.684,-79.913,-175.786,8.045,148.343
C06929=1216.607,396.931,-79.947,-175.785,8.048,148.344
C06930=1216.603,397.179,-79.982,-175.785,8.050,148.344
C06931=1216.599,397.426,-80.016,-175.784,8.053,148.345
C06932=1216.594,397.673,-80.050,-175.783,8.055,148.345
C06933=1216.590,397.921,-80.085,-175.783,8.057,148.345
C06934=1216.587,398.169,-80.119,-175.782,8.060,148.346
C06935=1216.583,398.417,-80.154,-175.782,8.062,148.346
C06936=1216.578,398.664,-80.188,-175.780,8.065,148.347
C06937=1216.574,398.911,-80.222,-175.780,8.067,148.347
C06938=1216.570,399.159,-80.257,-175.780,8.069,148.348
C06939=1216.566,399.407,-80.291,-175.779,8.072,148.348
C06940=1216.562,399.655,-80.325,-175.778,8.074,148.349
C06941=1216.558,399.902,-80.360,-175.778,8.077,148.349
C06942=1216.554,400.150,-80.395,-175.777,8.080,148.350
C06943=1216.550,400.397,-80.429,-175.777,8.082,148.350
C06944=1216.546,400.645,-80.463,-175.775,8.085,148.350
C06945=1216.542,400.893,-80.498,-175.775,8.087,148.351
C06946=1216.537,401.140,-80.532,-175.775,8.089,148.351
C06947=1216.534,401.387,-80.567,-175.774,8.092,148.352
C06948=1216.529,401.635,-80.602,-175.773,8.094,148.352
C06949=1216.526,401.883,-80.637,-175.773,8.096,148.353
C06950=1216.522,402.130,-80.670,-175.772,8.098,148.353
C06951=1216.518,402.378,-80.705,-175.772,8.101,148.354
C06952=1216.513,402.626,-80.740,-175.771,8.104,148.354
C06953=1216.509,402.874,-80.775,-175.771,8.106,148.355
C06954=1216.505,403.121,-80.808,-175.770,8.109,148.355
C06955=1216.501,403.368,-80.844,-175.769,8.111,148.356
C06956=1216.497,403.616,-80.879,-175.769,8.113,148.356
C06957=1216.493,403.863,-80.912,-175.769,8.115,148.356
C06958=1216.489,404.111,-80.947,-175.768,8.118,148.357
C06959=1216.485,404.358,-80.982,-175.767,8.120,148.357
C06960=1216.481,404.606,-81.017,-175.767,8.122,148.358
C06961=1216.477,404.853,-81.051,-175.766,8.124,148.358
C06962=1216.473,405.101,-81.086,-175.766,8.127,148.359
C06963=1216.469,405.348,-81.120,-175.765,8.129,148.359
C06964=1216.465,405.597,-81.155,-175.765,8.132,148.360
C06965=1216.460,405.843,-81.190,-175.764,8.134,148.360
C06966=1216.457,406.091,-81.225,-175.763,8.137,148.361
C06967=1216.453,406.339,-81.259,-175.763,8.139,148.361
C06968=1216.449,406.587,-81.294,-175.762,8.141,148.362
C06969=1216.444,406.834,-81.328,-175.762,8.143,148.362
C06970=1216.441,407.081,-81.363,-175.762,8.145,148.362
C06971=1216.437,407.329,-81.398,-175.761,8.148,148.363
C06972=1216.433,407.577,-81.433,-175.760,8.150,148.363
C06973=1216.428,407.824,-81.467,-175.760,8.153,148.364
C06974=1216.424,408.072,-81.503,-175.759,8.154,148.364
C06975=1216.421,408.319,-81.537,-175.759,8.157,148.365
C06976=1216.417,408.567,-81.571,-175.758,8.159,148.365
C06977=1216.412,408.814,-81.607,-175.758,8.162,148.366
C06978=1216.408,409.062,-81.641,-175.757,8.164,148.366
C06979=1216.404,409.309,-81.676,-175.757,8.166,148.367
C06980=1216.401,409.557,-81.710,-175.756,8.168,148.367
C06981=1216.396,409.804,-81.745,-175.756,8.170,148.367
C06982=1216.392,410.052,-81.780,-175.755,8.172,148.368
C06983=1216.388,410.300,-81.815,-175.755,8.175,148.368
C06984=1216.384,410.547,-81.850,-175.754,8.177,148.369
C06985=1216.380,410.794,-81.885,-175.754,8.180,148.369
C06986=1216.376,411.042,-81.919,-175.753,8.182,148.370
C06987=1216.372,411.289,-81.954,-175.753,8.184,148.370
C06988=1216.368,411.537,-81.989,-175.753,8.186,148.371
C06989=1216.364,411.785,-82.023,-175.752,8.188,148.371
C06990=1216.360,412.032,-82.059,-175.752,8.190,148.372
C06991=1216.356,412.280,-82.094,-175.751,8.192,148.372
C06992=1216.352,412.527,-82.129,-175.751,8.195,148.372
C06993=1216.348,412.775,-82.163,-175.750,8.197,148.373
C06994=1216.344,413.022,-82.198,-175.750,8.200,148.373
C06995=1216.340,413.270,-82.233,-175.749,8.202,148.374
C06996=1216.336,413.517,-82.268,-175.749,8.204,148.374
C06997=1216.332,413.765,-82.302,-175.748,8.206,148.375
C06998=1216.327,414.012,-82.338,-175.748,8.208,148.375
C06999=1216.323,414.260,-82.372,-175.747,8.210,148.375
C07000=1216.319,414.507,-82.408,-175.747,8.212,148.376
C07001=1216.316,414.755,-82.442,-175.746,8.214,148.376
C07002=1216.312,415.003,-82.477,-175.746,8.217,148.377
C07003=1216.308,415.250,-82.512,-175.746,8.219,148.377
C07004=1216.304,415.480,-82.545,-175.745,8.221,148.378
C07005=1216.300,415.710,-82.577,-175.745,8.223,148.378
C07006=1216.296,415.940,-82.609,-175.744,8.225,148.378
C07007=1216.293,416.170,-82.642,-175.744,8.227,148.379
C07008=1216.289,416.400,-82.675,-175.744,8.228,148.379
C07009=1216.285,416.631,-82.707,-175.743,8.230,148.380
C07010=1216.283,416.861,-82.739,-175.743,8.233,148.380
C07011=1216.284,417.091,-82.771,-175.742,8.235,148.380
C07012=1215.862,417.090,-82.807,-175.746,8.245,148.384
C07013=1215.860,416.860,-82.774,-175.746,8.243,148.384
C07014=1215.863,416.628,-82.742,-175.746,8.241,148.383
C07015=1215.867,416.396,-82.709,-175.747,8.239,148.383
C07016=1215.871,416.165,-82.677,-175.747,8.237,148.382
C07017=1215.874,415.934,-82.644,-175.747,8.236,148.382
C07018=1215.878,415.702,-82.611,-175.748,8.234,148.382
C07019=1215.882,415.471,-82.579,-175.748,8.231,148.381
C07020=1215.885,415.239,-82.546,-175.749,8.229,148.381
C07021=1215.890,414.992,-82.511,-175.749,8.227,148.380
C07022=1215.894,414.744,-82.476,-175.750,8.225,148.380
C07023=1215.898,414.497,-82.441,-175.750,8.223,148.380
C07024=1215.902,414.249,-82.406,-175.751,8.221,148.379
C07025=1215.906,414.001,-82.371,-175.751,8.219,148.379
C07026=1215.910,413.754,-82.336,-175.752,8.217,148.378
C07027=1215.913,413.507,-82.302,-175.752,8.214,148.378
C07028=1215.918,413.259,-82.267,-175.752,8.212,148.377
C07029=1215.922,413.012,-82.232,-175.753,8.210,148.377
C07030=1215.926,412.764,-82.197,-175.754,8.207,148.377
C07031=1215.930,412.516,-82.162,-175.754,8.205,148.376
C07032=1215.934,412.269,-82.127,-175.755,8.203,148.376
C07033=1215.938,412.021,-82.092,-175.755,8.201,148.375
C07034=1215.943,411.774,-82.057,-175.755,8.199,148.375
C07035=1215.946,411.527,-82.023,-175.756,8.197,148.374
C07036=1215.950,411.279,-81.988,-175.756,8.194,148.374
C07037=1215.954,411.032,-81.953,-175.757,8.192,148.373
C07038=1215.958,410.784,-81.918,-175.757,8.190,148.373
C07039=1215.963,410.536,-81.883,-175.757,8.188,148.372
C07040=1215.966,410.289,-81.848,-175.758,8.185,148.372
C07041=1215.970,410.042,-81.814,-175.759,8.183,148.372
C07042=1215.974,409.793,-81.779,-175.759,8.181,148.371
C07043=1215.978,409.547,-81.744,-175.760,8.179,148.371
C07044=1215.982,409.299,-81.709,-175.760,8.176,148.370
C07045=1215.987,409.051,-81.675,-175.760,8.174,148.370
C07046=1215.991,408.804,-81.639,-175.761,8.172,148.369
C07047=1215.994,408.557,-81.605,-175.762,8.169,148.369
C07048=1215.998,408.308,-81.571,-175.762,8.167,148.368
C07049=1216.003,408.061,-81.536,-175.763,8.165,148.368
C07050=1216.007,407.813,-81.500,-175.763,8.163,148.367
C07051=1216.011,407.566,-81.466,-175.763,8.161,148.367
C07052=1216.014,407.318,-81.432,-175.764,8.159,148.367
C07053=1216.019,407.071,-81.397,-175.765,8.155,148.366
C07054=1216.023,406.823,-81.362,-175.765,8.154,148.366
C07055=1216.027,406.576,-81.327,-175.765,8.151,148.365
C07056=1216.031,406.328,-81.292,-175.766,8.149,148.365
C07057=1216.035,406.081,-81.258,-175.766,8.147,148.364
C07058=1216.039,405.833,-81.223,-175.767,8.144,148.364
C07059=1216.043,405.586,-81.189,-175.768,8.142,148.363
C07060=1216.047,405.338,-81.154,-175.768,8.140,148.363
C07061=1216.051,405.091,-81.120,-175.768,8.138,148.362
C07062=1216.055,404.843,-81.084,-175.769,8.136,148.362
C07063=1216.059,404.596,-81.050,-175.770,8.133,148.361
C07064=1216.063,404.347,-81.015,-175.770,8.130,148.361
C07065=1216.068,404.100,-80.981,-175.771,8.128,148.361
C07066=1216.071,403.852,-80.946,-175.771,8.126,148.360
C07067=1216.075,403.605,-80.911,-175.772,8.123,148.360
C07068=1216.079,403.357,-80.876,-175.772,8.121,148.359
C07069=1216.083,403.110,-80.842,-175.773,8.119,148.359
C07070=1216.087,402.862,-80.808,-175.774,8.116,148.358
C07071=1216.092,402.615,-80.773,-175.774,8.114,148.358
C07072=1216.096,402.367,-80.738,-175.775,8.112,148.357
C07073=1216.099,402.120,-80.704,-175.775,8.110,148.357
C07074=1216.104,401.873,-80.669,-175.776,8.107,148.356
C07075=1216.108,401.625,-80.634,-175.777,8.105,148.356
C07076=1216.112,401.377,-80.600,-175.777,8.102,148.356
C07077=1216.115,401.129,-80.566,-175.778,8.100,148.355
C07078=1216.120,400.882,-80.531,-175.778,8.097,148.355
C07079=1216.124,400.634,-80.496,-175.778,8.095,148.354
C07080=1216.128,400.387,-80.463,-175.780,8.092,148.354
C07081=1216.132,400.139,-80.428,-175.780,8.090,148.353
C07082=1216.136,399.891,-80.393,-175.780,8.088,148.353
C07083=1216.140,399.645,-80.359,-175.781,8.085,148.352
C07084=1216.144,399.397,-80.324,-175.782,8.083,148.352
C07085=1216.148,399.149,-80.289,-175.782,8.081,148.351
C07086=1216.152,398.901,-80.255,-175.783,8.078,148.351
C07087=1216.156,398.654,-80.221,-175.783,8.075,148.350
C07088=1216.160,398.406,-80.186,-175.785,8.073,148.350
C07089=1216.164,398.159,-80.152,-175.785,8.070,148.349
C07090=1216.169,397.911,-80.118,-175.785,8.068,148.349
C07091=1216.173,397.663,-80.083,-175.786,8.065,148.348
C07092=1216.176,397.416,-80.049,-175.787,8.063,148.348
C07093=1216.180,397.168,-80.014,-175.788,8.060,148.348
C07094=1216.185,396.920,-79.980,-175.788,8.058,148.347
C07095=1216.189,396.673,-79.946,-175.789,8.055,148.347
C07096=1216.193,396.425,-79.911,-175.790,8.053,148.346
C07097=1216.197,396.178,-79.876,-175.790,8.051,148.346
C07098=1216.201,395.930,-79.842,-175.791,8.048,148.345
C07099=1216.205,395.683,-79.808,-175.791,8.046,148.345
C07100=1216.209,395.435,-79.774,-175.792,8.043,148.344
C07101=1216.213,395.187,-79.739,-175.793,8.041,148.344
C07102=1216.218,394.940,-79.704,-175.794,8.038,148.343
C07103=1216.221,394.692,-79.670,-175.794,8.036,148.343
C07104=1216.225,394.445,-79.636,-175.795,8.033,148.343
C07105=1216.229,394.198,-79.602,-175.796,8.031,148.342
C07106=1216.233,393.949,-79.567,-175.797,8.028,148.342
C07107=1216.238,393.701,-79.533,-175.797,8.026,148.341
C07108=1216.242,393.454,-79.499,-175.798,8.023,148.341
C07109=1216.246,393.172,-79.460,-175.799,8.020,148.340
C07110=1216.251,392.890,-79.421,-175.800,8.017,148.340
C07111=1216.255,392.608,-79.382,-175.801,8.014,148.339
C07112=1216.260,392.327,-79.343,-175.801,8.012,148.339
C07113=1216.264,392.078,-79.309,-175.802,8.009,148.338
C07114=1216.268,391.831,-79.275,-175.803,8.006,148.338
C07115=1216.272,391.583,-79.240,-175.803,8.003,148.337
C07116=1216.276,391.336,-79.206,-175.805,8.001,148.337
C07117=1216.281,391.088,-79.171,-175.805,7.998,148.336
C07118=1216.284,390.840,-79.137,-175.806,7.996,148.336
C07119=1216.289,390.593,-79.103,-175.807,7.994,148.336
C07120=1216.293,390.345,-79.070,-175.807,7.990,148.335
C07121=1216.297,390.097,-79.035,-175.809,7.988,148.335
C07122=1216.301,389.850,-79.001,-175.809,7.985,148.334
C07123=1216.305,389.603,-78.966,-175.810,7.983,148.334
C07124=1216.308,389.355,-78.932,-175.811,7.980,148.333
C07125=1216.313,389.107,-78.898,-175.811,7.977,148.333
C07126=1216.317,388.860,-78.865,-175.813,7.975,148.332
C07127=1216.321,388.612,-78.830,-175.813,7.972,148.332
C07128=1216.325,388.364,-78.796,-175.814,7.970,148.331
C07129=1216.330,388.116,-78.762,-175.815,7.967,148.331
C07130=1216.333,387.869,-78.728,-175.816,7.964,148.330
C07131=1216.338,387.621,-78.693,-175.816,7.962,148.330
C07132=1216.341,387.374,-78.659,-175.818,7.959,148.330
C07133=1216.345,387.126,-78.626,-175.818,7.956,148.329
C07134=1216.349,386.878,-78.592,-175.819,7.954,148.329
C07135=1216.353,386.631,-78.558,-175.820,7.951,148.328
C07136=1216.358,386.383,-78.524,-175.821,7.948,148.328
C07137=1216.361,386.135,-78.490,-175.822,7.945,148.327
C07138=1216.366,385.888,-78.455,-175.823,7.943,148.327
C07139=1216.370,385.641,-78.421,-175.824,7.940,148.326
C07140=1216.374,385.392,-78.387,-175.825,7.937,148.326
C07141=1216.378,385.145,-78.353,-175.826,7.934,148.326
C07142=1216.382,384.898,-78.319,-175.827,7.932,148.325
C07143=1216.387,384.650,-78.286,-175.827,7.929,148.325
C07144=1216.390,384.402,-78.251,-175.829,7.926,148.324
C07145=1216.395,384.154,-78.218,-175.830,7.924,148.324
C07146=1216.399,383.907,-78.184,-175.830,7.922,148.323
C07147=1216.402,383.660,-78.150,-175.831,7.918,148.323
C07148=1216.407,383.411,-78.116,-175.832,7.916,148.322
C07149=1216.410,383.164,-78.082,-175.833,7.913,148.322
C07150=1216.415,382.916,-78.048,-175.835,7.910,148.322
C07151=1216.419,382.669,-78.014,-175.835,7.908,148.321
C07152=1216.422,382.421,-77.980,-175.836,7.905,148.321
C07153=1216.427,382.173,-77.946,-175.837,7.902,148.320
C07154=1216.431,381.926,-77.912,-175.838,7.899,148.320
C07155=1216.435,381.678,-77.879,-175.839,7.896,148.319
C07156=1216.439,381.430,-77.845,-175.840,7.893,148.319
C07157=1216.443,381.182,-77.811,-175.841,7.891,148.319
C07158=1216.447,380.935,-77.777,-175.842,7.889,148.318
C07159=1216.452,380.687,-77.744,-175.843,7.886,148.318
C07160=1216.455,380.439,-77.709,-175.845,7.883,148.317
C07161=1216.459,380.191,-77.676,-175.845,7.880,148.317
C07162=1216.464,379.944,-77.642,-175.846,7.877,148.316
C07163=1216.468,379.696,-77.609,-175.848,7.874,148.316
C07164=1216.472,379.449,-77.575,-175.849,7.871,148.316
C07165=1216.476,379.200,-77.541,-175.850,7.869,148.315
C07166=1216.480,378.953,-77.507,-175.851,7.866,148.315
C07167=1216.484,378.706,-77.474,-175.852,7.864,148.315
C07168=1216.489,378.458,-77.439,-175.853,7.861,148.314
C07169=1216.493,378.210,-77.406,-175.854,7.858,148.314
C07170=1216.496,377.963,-77.372,-175.855,7.855,148.313
C07171=1216.500,377.715,-77.339,-175.856,7.852,148.313
C07172=1216.505,377.467,-77.305,-175.857,7.849,148.312
C07173=1216.509,377.220,-77.271,-175.859,7.847,148.312
C07174=1216.513,376.972,-77.238,-175.860,7.844,148.312
C07175=1216.516,376.724,-77.204,-175.861,7.841,148.311
C07176=1216.521,376.476,-77.170,-175.862,7.838,148.311
C07177=1216.525,376.228,-77.137,-175.863,7.835,148.310
C07178=1216.529,375.981,-77.103,-175.865,7.833,148.310
C07179=1216.533,375.734,-77.070,-175.866,7.830,148.310
C07180=1216.538,375.486,-77.036,-175.867,7.827,148.309
C07181=1216.541,375.238,-77.002,-175.868,7.824,148.309
C07182=1216.546,374.990,-76.969,-175.869,7.821,148.308
C07183=1216.550,374.742,-76.935,-175.870,7.818,148.308
C07184=1216.554,374.495,-76.902,-175.872,7.816,148.308
C07185=1216.558,374.247,-76.868,-175.873,7.813,148.307
C07186=1216.563,373.999,-76.835,-175.874,7.810,148.307
C07187=1216.566,373.752,-76.800,-175.875,7.807,148.306
C07188=1216.570,373.504,-76.767,-175.876,7.804,148.306
C07189=1216.574,373.256,-76.734,-175.878,7.802,148.306
C07190=1216.578,373.008,-76.701,-175.879,7.799,148.306
C07191=1216.583,372.761,-76.666,-175.881,7.795,148.305
C07192=1216.587,372.513,-76.633,-175.882,7.793,148.305
C07193=1216.591,372.266,-76.600,-175.883,7.790,148.304
C07194=1216.595,372.018,-76.567,-175.885,7.787,148.304
C07195=1216.599,371.769,-76.533,-175.886,7.784,148.303
C07196=1216.603,371.522,-76.500,-175.887,7.781,148.303
C07197=1216.607,371.275,-76.466,-175.888,7.778,148.303
C07198=1216.611,371.027,-76.433,-175.890,7.776,148.303
C07199=1216.616,370.779,-76.400,-175.891,7.773,148.302
C07200=1216.620,370.531,-76.366,-175.892,7.770,148.302
C07201=1216.624,370.283,-76.333,-175.894,7.767,148.301
C07202=1216.628,370.036,-76.299,-175.895,7.764,148.301
C07203=1216.632,369.788,-76.266,-175.897,7.761,148.301
C07204=1216.636,369.541,-76.233,-175.898,7.759,148.300
C07205=1216.640,369.293,-76.200,-175.899,7.756,148.300
C07206=1216.644,369.045,-76.166,-175.900,7.753,148.300
C07207=1216.648,368.797,-76.133,-175.902,7.750,148.299
C07208=1216.652,368.549,-76.100,-175.904,7.747,148.299
C07209=1216.656,368.301,-76.067,-175.905,7.744,148.298
C07210=1216.660,368.054,-76.034,-175.906,7.741,148.298
C07211=1216.664,367.806,-76.001,-175.908,7.739,148.298
C07212=1216.669,367.558,-75.967,-175.909,7.736,148.298
C07213=1216.674,367.278,-75.929,-175.911,7.732,148.297
C07214=1216.679,366.999,-75.892,-175.912,7.728,148.297
C07215=1216.683,366.718,-75.854,-175.914,7.726,148.296
C07216=1216.687,366.438,-75.817,-175.916,7.722,148.296
C07217=1216.692,366.191,-75.784,-175.917,7.719,148.296
C07218=1216.696,365.943,-75.751,-175.919,7.717,148.295
C07219=1216.700,365.695,-75.718,-175.920,7.713,148.295
C07220=1216.704,365.447,-75.684,-175.921,7.710,148.295
C07221=1216.708,365.200,-75.651,-175.923,7.708,148.294
C07222=1216.712,364.952,-75.618,-175.924,7.705,148.294
C07223=1216.716,364.704,-75.585,-175.926,7.702,148.294
C07224=1216.721,364.456,-75.552,-175.928,7.699,148.293
C07225=1216.725,364.209,-75.519,-175.929,7.696,148.293
C07226=1216.729,363.961,-75.486,-175.930,7.694,148.293
C07227=1216.733,363.713,-75.452,-175.932,7.690,148.292
C07228=1216.736,363.466,-75.420,-175.934,7.687,148.292
C07229=1216.741,363.217,-75.387,-175.935,7.685,148.292
C07230=1216.745,362.970,-75.354,-175.937,7.682,148.292
C07231=1216.749,362.722,-75.321,-175.938,7.678,148.291
C07232=1216.753,362.474,-75.288,-175.940,7.676,148.291
C07233=1216.757,362.227,-75.255,-175.941,7.673,148.291
C07234=1216.762,361.979,-75.222,-175.943,7.670,148.290
C07235=1216.766,361.730,-75.189,-175.945,7.667,148.290
C07236=1216.770,361.483,-75.156,-175.946,7.664,148.290
C07237=1216.774,361.235,-75.123,-175.947,7.662,148.289
C07238=1216.778,360.988,-75.090,-175.950,7.658,148.289
C07239=1216.782,360.740,-75.057,-175.951,7.655,148.289
C07240=1216.786,360.491,-75.025,-175.952,7.653,148.289
C07241=1216.790,360.244,-74.992,-175.955,7.650,148.288
C07242=1216.795,359.996,-74.958,-175.956,7.647,148.288
C07243=1216.799,359.748,-74.925,-175.958,7.644,148.288
C07244=1216.802,359.500,-74.893,-175.959,7.641,148.287
C07245=1216.806,359.253,-74.860,-175.961,7.638,148.287
C07246=1216.811,359.005,-74.827,-175.963,7.636,148.287
C07247=1216.815,358.756,-74.795,-175.964,7.632,148.286
C07248=1216.820,358.509,-74.762,-175.966,7.629,148.286
C07249=1216.823,358.262,-74.729,-175.968,7.627,148.286
C07250=1216.828,358.014,-74.697,-175.969,7.623,148.286
C07251=1216.832,357.766,-74.664,-175.971,7.621,148.285
C07252=1216.836,357.518,-74.631,-175.973,7.618,148.285
C07253=1216.840,357.270,-74.599,-175.974,7.614,148.285
C07254=1216.844,357.022,-74.566,-175.976,7.612,148.285
C07255=1216.848,356.774,-74.533,-175.978,7.609,148.284
C07256=1216.852,356.526,-74.500,-175.979,7.606,148.284
C07257=1216.856,356.279,-74.467,-175.981,7.603,148.284
C07258=1216.861,356.031,-74.435,-175.983,7.601,148.284
C07259=1216.865,355.784,-74.402,-175.985,7.597,148.283
C07260=1216.869,355.535,-74.370,-175.986,7.595,148.283
C07261=1216.873,355.288,-74.337,-175.988,7.591,148.283
C07262=1216.877,355.039,-74.305,-175.990,7.589,148.283
C07263=1216.881,354.792,-74.272,-175.991,7.586,148.282
C07264=1216.885,354.544,-74.240,-175.993,7.582,148.282
C07265=1216.890,354.297,-74.207,-175.995,7.580,148.282
C07266=1216.894,354.048,-74.174,-175.997,7.577,148.282
C07267=1216.898,353.801,-74.142,-175.999,7.574,148.281
C07268=1216.902,353.553,-74.109,-176.000,7.572,148.281
C07269=1216.906,353.305,-74.076,-176.002,7.568,148.281
C07270=1216.910,353.057,-74.044,-176.004,7.565,148.281
C07271=1216.915,352.810,-74.012,-176.005,7.563,148.280
C07272=1216.919,352.561,-73.979,-176.008,7.560,148.280
C07273=1216.923,352.313,-73.947,-176.009,7.557,148.280
C07274=1216.927,352.066,-73.914,-176.011,7.555,148.280
C07275=1216.931,351.817,-73.882,-176.013,7.551,148.280
C07276=1216.935,351.570,-73.849,-176.014,7.548,148.279
C07277=1216.940,351.322,-73.817,-176.016,7.545,148.279
C07278=1216.944,351.074,-73.785,-176.018,7.542,148.279
C07279=1216.948,350.826,-73.752,-176.020,7.540,148.279
C07280=1216.952,350.578,-73.720,-176.022,7.537,148.278
C07281=1216.956,350.331,-73.688,-176.024,7.534,148.278
C07282=1216.961,350.083,-73.655,-176.026,7.531,148.278
C07283=1216.964,349.835,-73.623,-176.027,7.528,148.278
C07284=1216.969,349.587,-73.591,-176.029,7.526,148.278
C07285=1216.972,349.339,-73.558,-176.031,7.522,148.277
C07286=1216.977,349.092,-73.526,-176.033,7.520,148.277
C07287=1216.981,348.844,-73.494,-176.035,7.516,148.277
C07288=1216.985,348.595,-73.462,-176.037,7.514,148.277
C07289=1216.989,348.347,-73.429,-176.038,7.511,148.277
C07290=1216.994,348.100,-73.397,-176.041,7.508,148.276
C07291=1216.998,347.852,-73.365,-176.042,7.506,148.276
C07292=1217.002,347.604,-73.333,-176.044,7.502,148.276
C07293=1217.006,347.355,-73.301,-176.046,7.500,148.276
C07294=1217.010,347.109,-73.268,-176.048,7.497,148.276
C07295=1217.015,346.860,-73.236,-176.050,7.494,148.275
C07296=1217.019,346.612,-73.204,-176.051,7.491,148.275
C07297=1217.023,346.365,-73.173,-176.054,7.488,148.275
C07298=1217.027,346.117,-73.140,-176.055,7.485,148.275
C07299=1217.031,345.869,-73.108,-176.058,7.482,148.275
C07300=1217.035,345.620,-73.076,-176.059,7.479,148.274
C07301=1217.039,345.373,-73.044,-176.061,7.477,148.274
C07302=1217.044,345.125,-73.011,-176.063,7.474,148.274
C07303=1217.048,344.877,-72.979,-176.065,7.471,148.274
